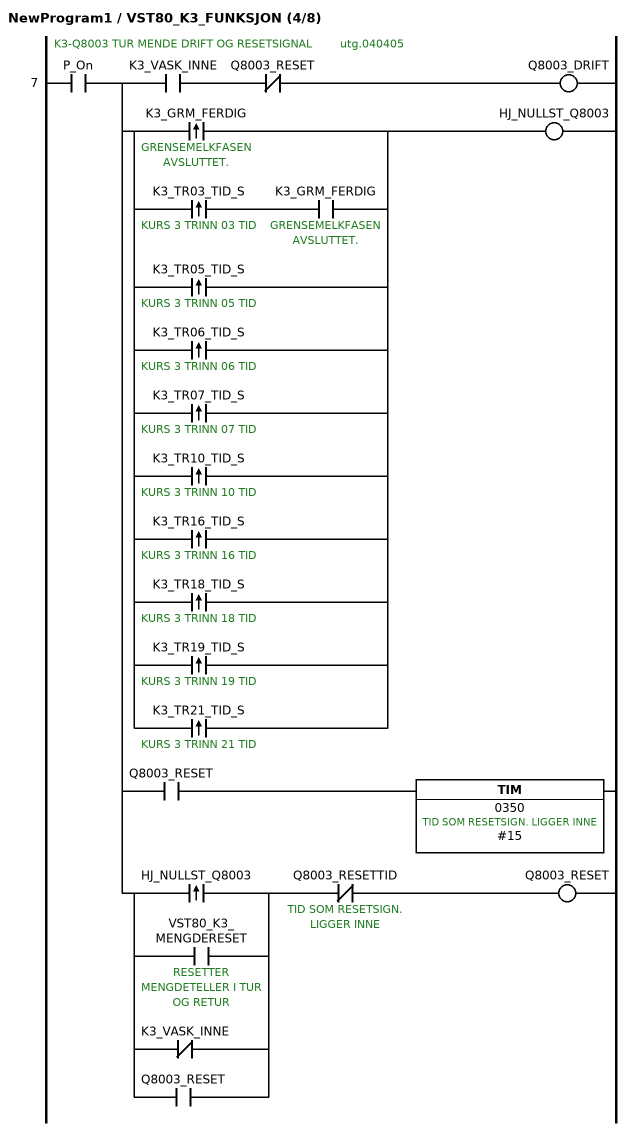
; [picture p360: NewProgram1 / VST80_K3_FUNKSJON, rungs 7-7]
; rung 7: K3-Q8003 TUR MENDE DRIFT OG RESETSIGNAL        utg.040405
LD P_On
OUT TR0
AND K3_VASK_INNE
ANDNOT Q8003_RESET
OUT Q8003_DRIFT
LD TR0
@LD K3_GRM_FERDIG  ; GRENSEMELKFASEN AVSLUTTET.
@LD K3_TR03_TID_S  ; KURS 3 TRINN 03 TID
AND K3_GRM_FERDIG  ; GRENSEMELKFASEN AVSLUTTET.
ORLD
@OR K3_TR05_TID_S  ; KURS 3 TRINN 05 TID
@OR K3_TR06_TID_S  ; KURS 3 TRINN 06 TID
@OR K3_TR07_TID_S  ; KURS 3 TRINN 07 TID
@OR K3_TR10_TID_S  ; KURS 3 TRINN 10 TID
@OR K3_TR16_TID_S  ; KURS 3 TRINN 16 TID
@OR K3_TR18_TID_S  ; KURS 3 TRINN 18 TID
@OR K3_TR19_TID_S  ; KURS 3 TRINN 19 TID
@OR K3_TR21_TID_S  ; KURS 3 TRINN 21 TID
ANDLD
OUT HJ_NULLST_Q8003
LD TR0
AND Q8003_RESET
TIM 0350 #15  ; TID SOM RESETSIGN. LIGGER INNE
LD TR0
@LD HJ_NULLST_Q8003
OR VST80_K3_MENGDERESET  ; RESETTER MENGDETELLER I TUR OG RETUR
ORNOT K3_VASK_INNE
OR Q8003_RESET
ANDLD
ANDNOT Q8003_RESETTID  ; TID SOM RESETSIGN. LIGGER INNE
OUT Q8003_RESET

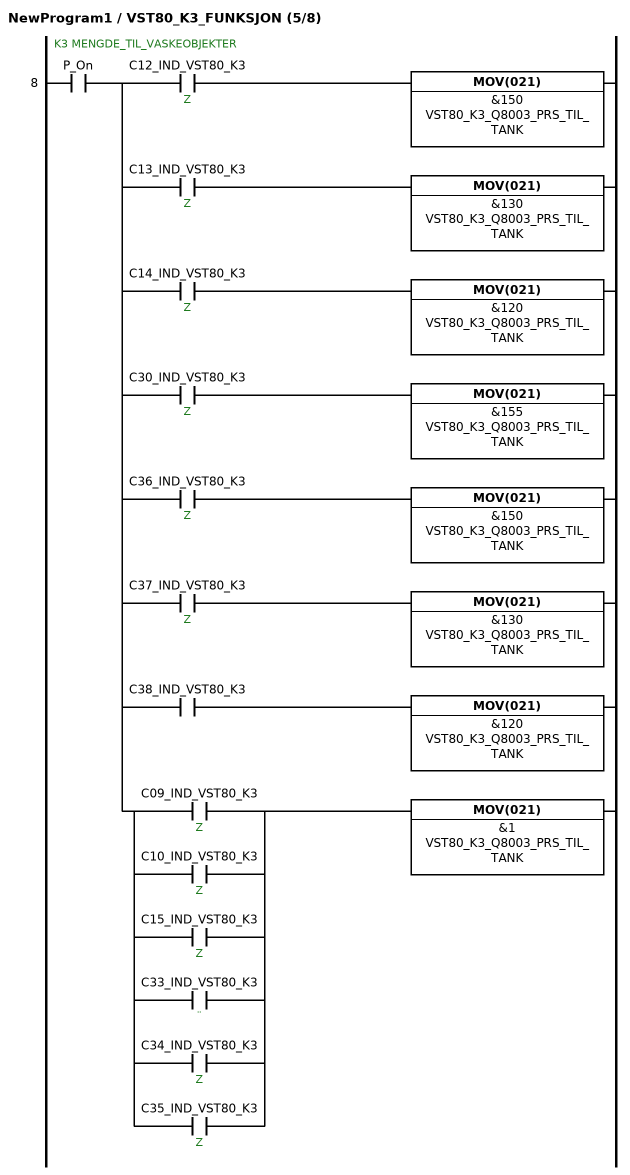
; rung 8: K3 MENGDE_TIL_VASKEOBJEKTER
LD P_On
OUT TR0
AND C12_IND_VST80_K3  ; Z
MOV(021) &150 VST80_K3_Q8003_PRS_TIL_TANK
LD TR0
AND C13_IND_VST80_K3  ; Z
MOV(021) &130 VST80_K3_Q8003_PRS_TIL_TANK
LD TR0
AND C14_IND_VST80_K3  ; Z
MOV(021) &120 VST80_K3_Q8003_PRS_TIL_TANK
LD TR0
AND C30_IND_VST80_K3  ; Z
MOV(021) &155 VST80_K3_Q8003_PRS_TIL_TANK
LD TR0
AND C36_IND_VST80_K3  ; Z
MOV(021) &150 VST80_K3_Q8003_PRS_TIL_TANK
LD TR0
AND C37_IND_VST80_K3  ; Z
MOV(021) &130 VST80_K3_Q8003_PRS_TIL_TANK
LD TR0
AND C38_IND_VST80_K3
MOV(021) &120 VST80_K3_Q8003_PRS_TIL_TANK
LD TR0
LD C09_IND_VST80_K3  ; Z
OR C10_IND_VST80_K3  ; Z
OR C15_IND_VST80_K3  ; Z
OR C33_IND_VST80_K3  ; ¨
OR C34_IND_VST80_K3  ; Z
OR C35_IND_VST80_K3  ; Z
ANDLD
MOV(021) &1 VST80_K3_Q8003_PRS_TIL_TANK

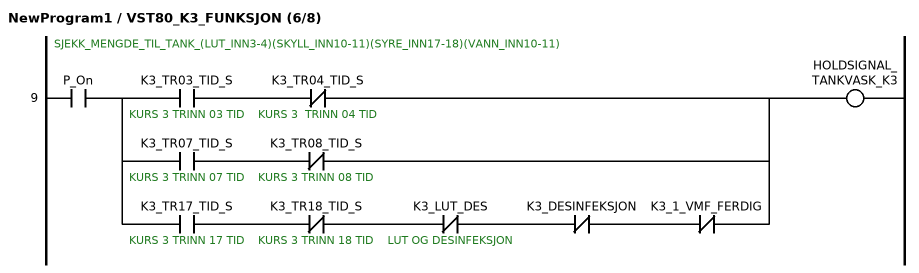
; rung 9: SJEKK_MENGDE_TIL_TANK_(LUT_INN3-4)(SKYLL_INN10-11)(SYRE_INN17-18)(VANN_INN10-11)
LD P_On
LD K3_TR03_TID_S  ; KURS 3 TRINN 03 TID
ANDNOT K3_TR04_TID_S  ; KURS 3  TRINN 04 TID
LD K3_TR07_TID_S  ; KURS 3 TRINN 07 TID
ANDNOT K3_TR08_TID_S  ; KURS 3 TRINN 08 TID
ORLD
LD K3_TR17_TID_S  ; KURS 3 TRINN 17 TID
ANDNOT K3_TR18_TID_S  ; KURS 3 TRINN 18 TID
ANDNOT K3_LUT_DES  ; LUT OG DESINFEKSJON
ANDNOT K3_DESINFEKSJON
ANDNOT K3_1_VMF_FERDIG
ORLD
ANDLD
OUT HOLDSIGNAL_TANKVASK_K3

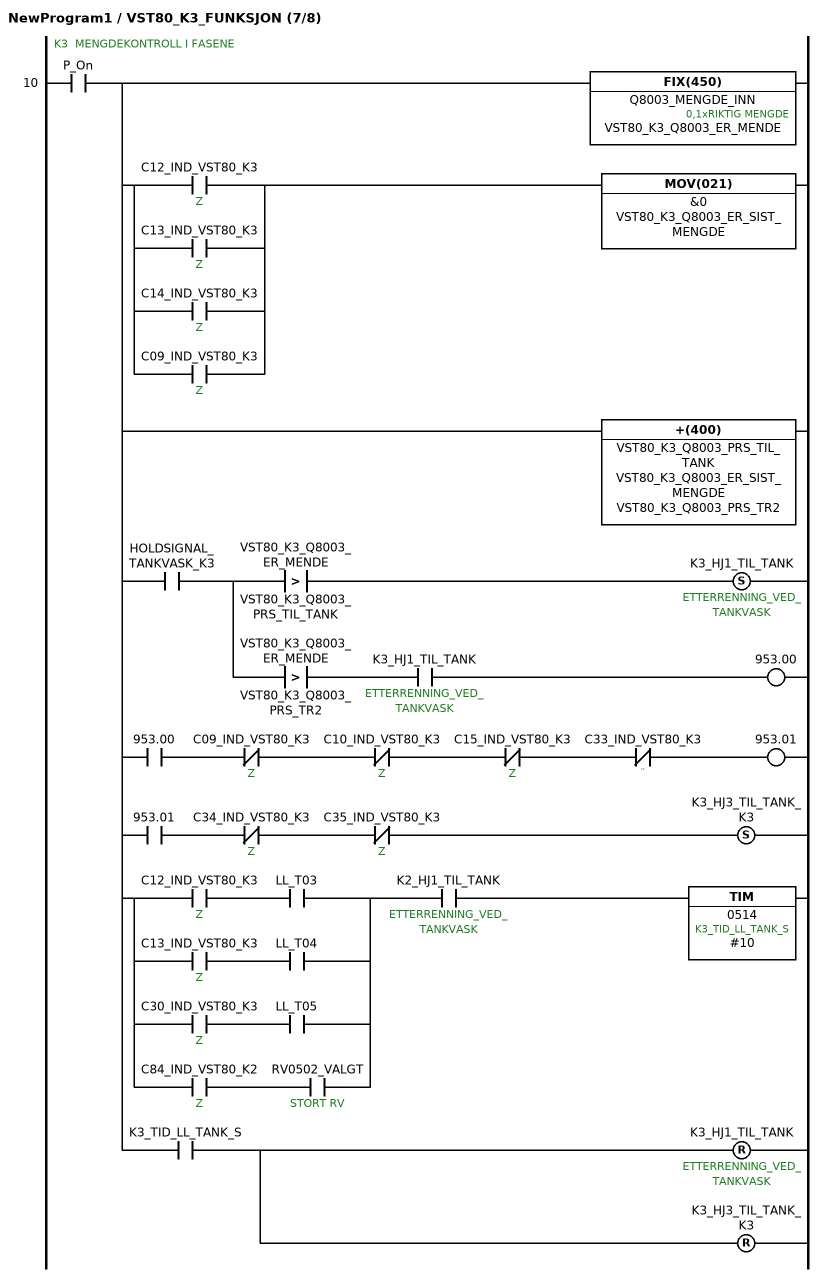
; rung 10: K3  MENGDEKONTROLL I FASENE
LD P_On
OUT TR0
FIX(450) Q8003_MENGDE_INN VST80_K3_Q8003_ER_MENDE  ; 0,1xRIKTIG MENGDE
LD C12_IND_VST80_K3  ; Z
OR C13_IND_VST80_K3  ; Z
OR C14_IND_VST80_K3  ; Z
OR C09_IND_VST80_K3  ; Z
ANDLD
MOV(021) &0 VST80_K3_Q8003_ER_SIST_MENGDE
LD TR0
+(400) VST80_K3_Q8003_PRS_TIL_TANK VST80_K3_Q8003_ER_SIST_MENGDE VST80_K3_Q8003_PRS_TR2
AND HOLDSIGNAL_TANKVASK_K3
OUT TR1
AND>(320) VST80_K3_Q8003_ER_MENDE VST80_K3_Q8003_PRS_TIL_TANK
SET K3_HJ1_TIL_TANK  ; ETTERRENNING_VED_TANKVASK
LD TR1
AND>(320) VST80_K3_Q8003_ER_MENDE VST80_K3_Q8003_PRS_TR2
AND K3_HJ1_TIL_TANK  ; ETTERRENNING_VED_TANKVASK
OUT 953.00
LD TR0
AND 953.00
ANDNOT C09_IND_VST80_K3  ; Z
ANDNOT C10_IND_VST80_K3  ; Z
ANDNOT C15_IND_VST80_K3  ; Z
ANDNOT C33_IND_VST80_K3  ; ¨
OUT 953.01
LD TR0
AND 953.01
ANDNOT C34_IND_VST80_K3  ; Z
ANDNOT C35_IND_VST80_K3  ; Z
SET K3_HJ3_TIL_TANK_K3
LD TR0
LD C12_IND_VST80_K3  ; Z
AND LL_T03
LD C13_IND_VST80_K3  ; Z
AND LL_T04
ORLD
LD C30_IND_VST80_K3  ; Z
AND LL_T05
ORLD
LD C84_IND_VST80_K2  ; Z
AND RV0502_VALGT  ; STORT RV
ORLD
ANDLD
AND K2_HJ1_TIL_TANK  ; ETTERRENNING_VED_TANKVASK
TIM 0514 #10  ; K3_TID_LL_TANK_S
LD TR0
AND K3_TID_LL_TANK_S
RSET K3_HJ1_TIL_TANK  ; ETTERRENNING_VED_TANKVASK
RSET K3_HJ3_TIL_TANK_K3

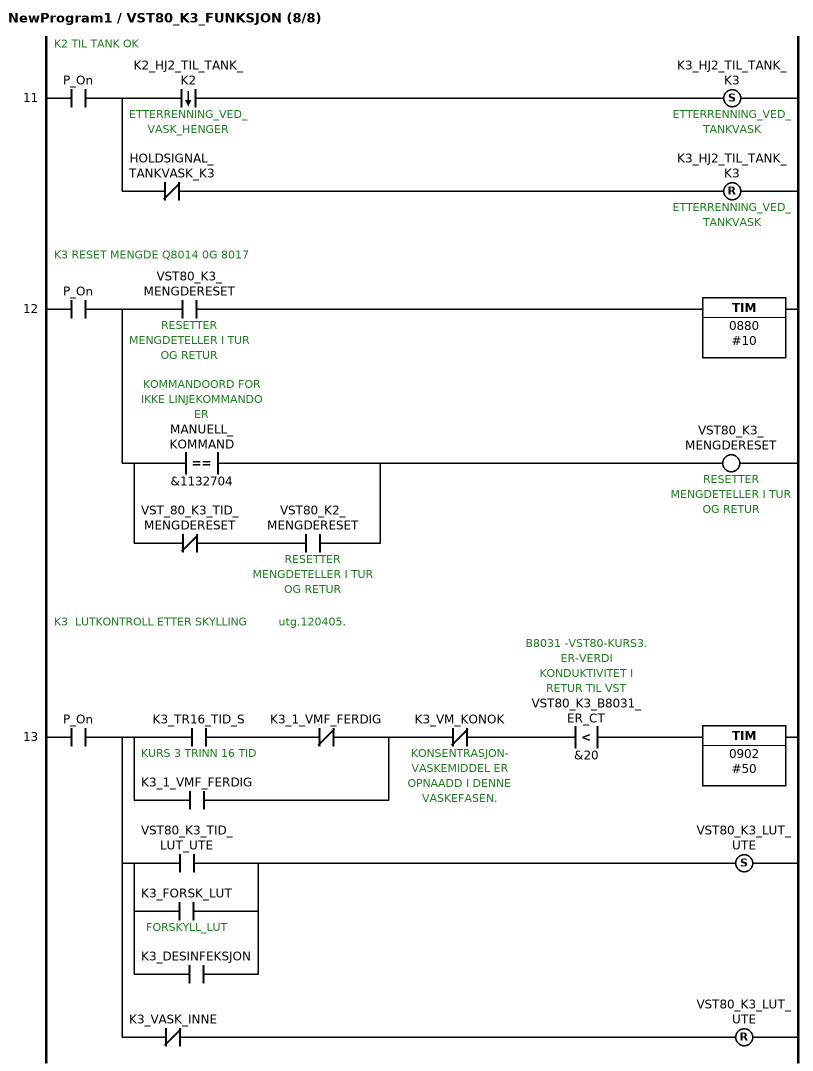
; rung 11: K2 TIL TANK OK
LD P_On
OUT TR0
%AND K2_HJ2_TIL_TANK_K2  ; ETTERRENNING_VED_VASK_HENGER
SET K3_HJ2_TIL_TANK_K3  ; ETTERRENNING_VED_TANKVASK
LD TR0
ANDNOT HOLDSIGNAL_TANKVASK_K3
RSET K3_HJ2_TIL_TANK_K3  ; ETTERRENNING_VED_TANKVASK
; rung 12: K3 RESET MENGDE Q8014 0G 8017
LD P_On
OUT TR0
AND VST80_K3_MENGDERESET  ; RESETTER MENGDETELLER I TUR OG RETUR
TIM 0880 #10
LD TR0
LD=L(301) MANUELL_KOMMAND &1132704  ; KOMMANDOORD FOR IKKE LINJEKOMMANDOER
LDNOT VST_80_K3_TID_MENGDERESET
AND VST80_K2_MENGDERESET  ; RESETTER MENGDETELLER I TUR OG RETUR
ORLD
ANDLD
OUT VST80_K3_MENGDERESET  ; RESETTER MENGDETELLER I TUR OG RETUR
; rung 13: K3  LUTKONTROLL ETTER SKYLLING         utg.120405.
LD P_On
OUT TR0
LD K3_TR16_TID_S  ; KURS 3 TRINN 16 TID
ANDNOT K3_1_VMF_FERDIG
OR K3_1_VMF_FERDIG
ANDLD
ANDNOT K3_VM_KONOK  ; KONSENTRASJON-VASKEMIDDEL ER OPNAADD I DENNE VASKEFASEN.
AND<(310) VST80_K3_B8031_ER_CT &20  ; B8031 -VST80-KURS3. ER-VERDI KONDUKTIVITET I RETUR TIL VST
TIM 0902 #50
LD TR0
LD VST80_K3_TID_LUT_UTE
OR K3_FORSK_LUT  ; FORSKYLL_LUT
OR K3_DESINFEKSJON
ANDLD
SET VST80_K3_LUT_UTE
LD TR0
ANDNOT K3_VASK_INNE
RSET VST80_K3_LUT_UTE
; rung 14: Ingen_kommentar_funnet

### Section VST80_K3_OBJEKTER
; Styring av objektene i kurs K1

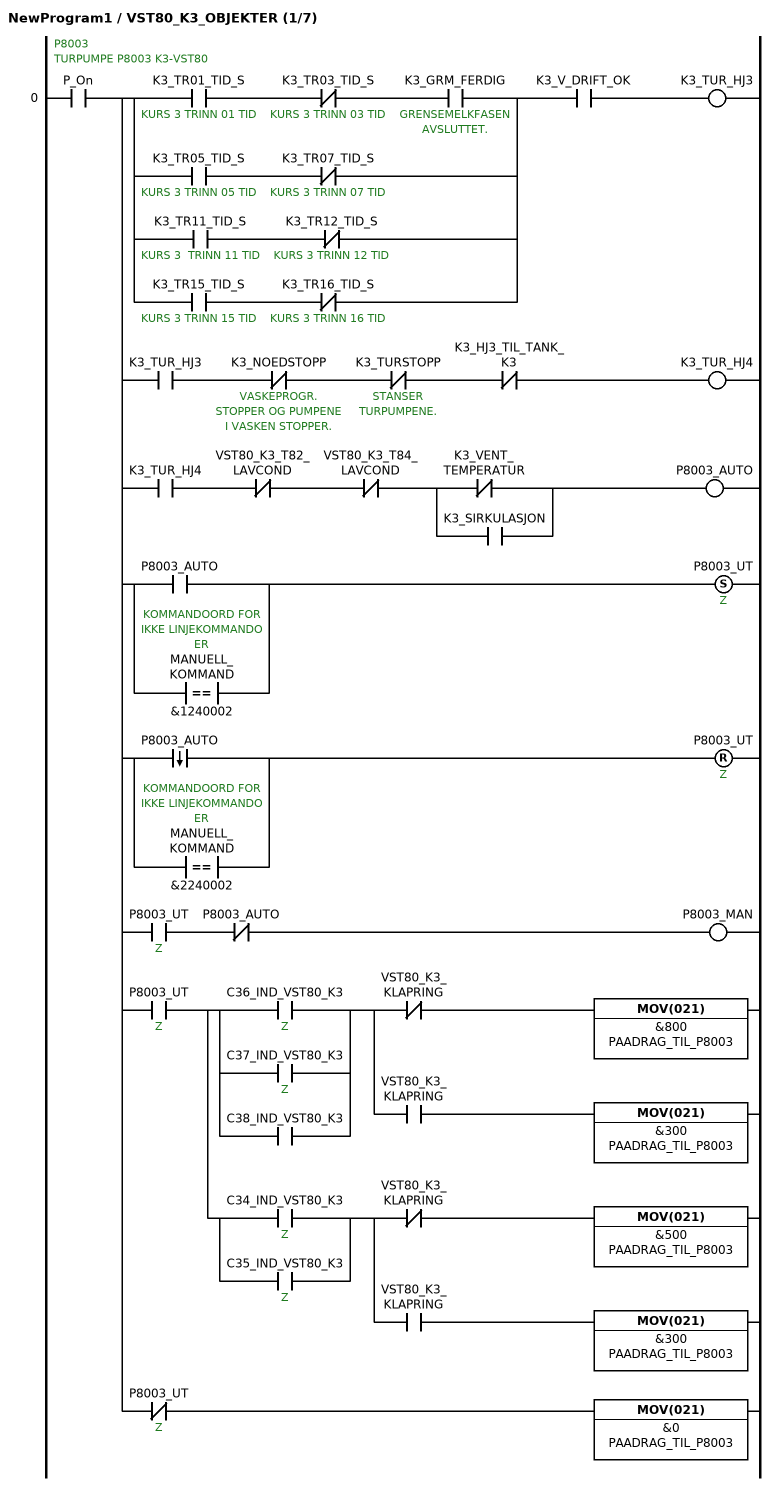
; rung 0: P8003 / TURPUMPE P8003 K3-VST80
LD P_On
OUT TR0
LD K3_TR01_TID_S  ; KURS 3 TRINN 01 TID
ANDNOT K3_TR03_TID_S  ; KURS 3 TRINN 03 TID
AND K3_GRM_FERDIG  ; GRENSEMELKFASEN AVSLUTTET.
LD K3_TR05_TID_S  ; KURS 3 TRINN 05 TID
ANDNOT K3_TR07_TID_S  ; KURS 3 TRINN 07 TID
ORLD
LD K3_TR11_TID_S  ; KURS 3  TRINN 11 TID
ANDNOT K3_TR12_TID_S  ; KURS 3 TRINN 12 TID
ORLD
LD K3_TR15_TID_S  ; KURS 3 TRINN 15 TID
ANDNOT K3_TR16_TID_S  ; KURS 3 TRINN 16 TID
ORLD
ANDLD
AND K3_V_DRIFT_OK
OUT K3_TUR_HJ3
LD TR0
AND K3_TUR_HJ3
ANDNOT K3_NOEDSTOPP  ; VASKEPROGR. STOPPER OG PUMPENE I VASKEN STOPPER.
ANDNOT K3_TURSTOPP  ; STANSER TURPUMPENE.
ANDNOT K3_HJ3_TIL_TANK_K3
OUT K3_TUR_HJ4
LD TR0
AND K3_TUR_HJ4
ANDNOT VST80_K3_T82_LAVCOND
ANDNOT VST80_K3_T84_LAVCOND
LDNOT K3_VENT_TEMPERATUR
OR K3_SIRKULASJON
ANDLD
OUT P8003_AUTO
LD TR0
LD P8003_AUTO
OR=L(301) MANUELL_KOMMAND &1240002  ; KOMMANDOORD FOR IKKE LINJEKOMMANDOER
ANDLD
SET P8003_UT  ; Z
LD TR0
%LD P8003_AUTO
OR=L(301) MANUELL_KOMMAND &2240002  ; KOMMANDOORD FOR IKKE LINJEKOMMANDOER
ANDLD
RSET P8003_UT  ; Z
LD TR0
AND P8003_UT  ; Z
ANDNOT P8003_AUTO
OUT P8003_MAN
LD TR0
AND P8003_UT  ; Z
OUT TR1
LD C36_IND_VST80_K3  ; Z
OR C37_IND_VST80_K3  ; Z
OR C38_IND_VST80_K3
ANDLD
OUT TR2
ANDNOT VST80_K3_KLAPRING
MOV(021) &800 PAADRAG_TIL_P8003
LD TR2
AND VST80_K3_KLAPRING
MOV(021) &300 PAADRAG_TIL_P8003
LD TR1
LD C34_IND_VST80_K3  ; Z
OR C35_IND_VST80_K3  ; Z
ANDLD
OUT TR1
ANDNOT VST80_K3_KLAPRING
MOV(021) &500 PAADRAG_TIL_P8003
LD TR1
AND VST80_K3_KLAPRING
MOV(021) &300 PAADRAG_TIL_P8003
LD TR0
ANDNOT P8003_UT  ; Z
MOV(021) &0 PAADRAG_TIL_P8003

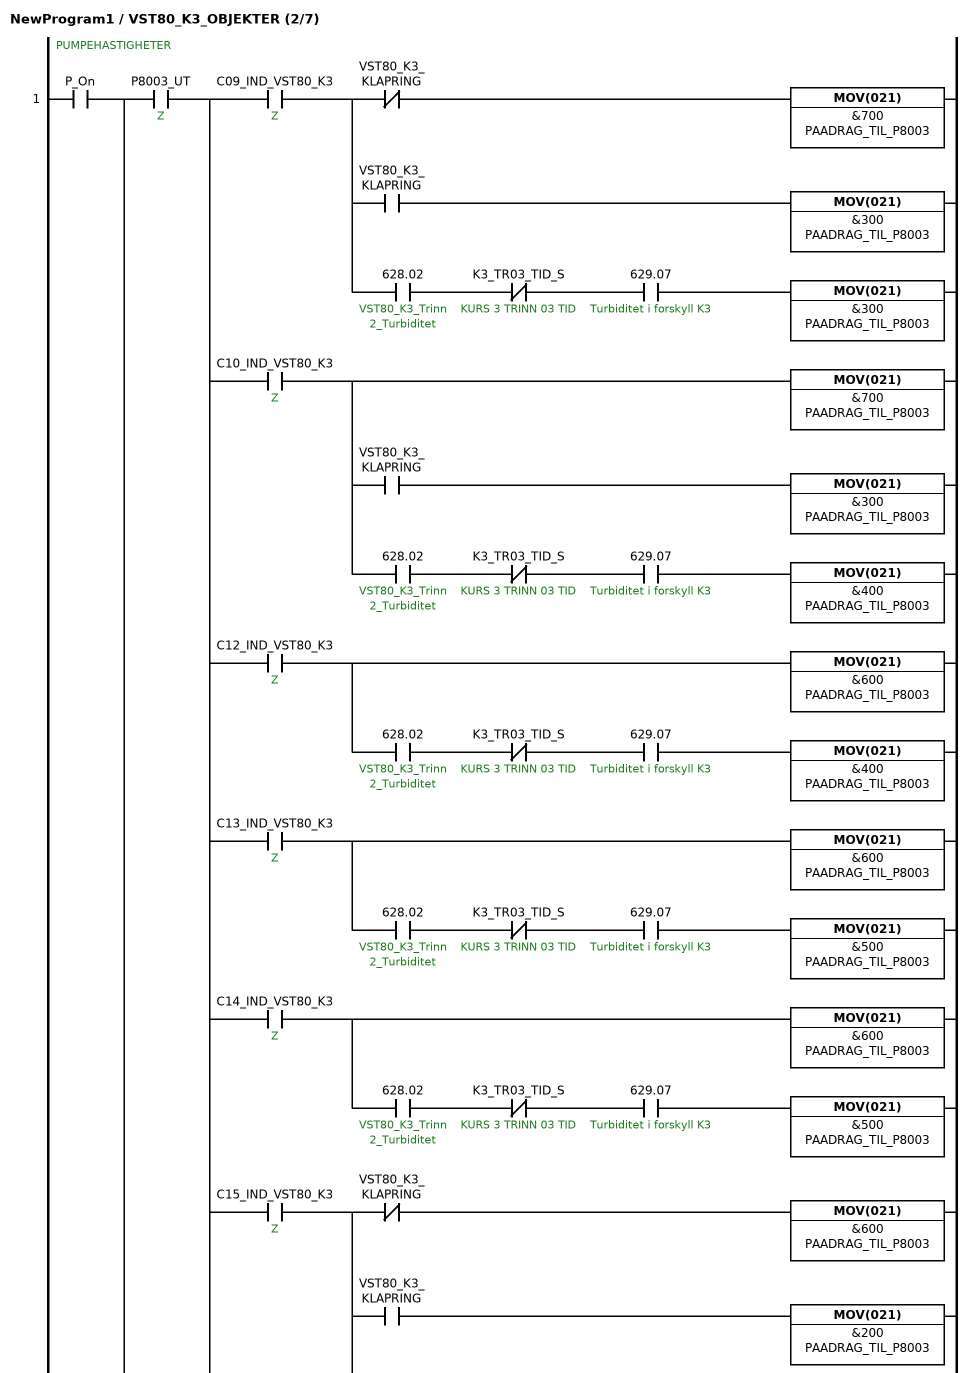

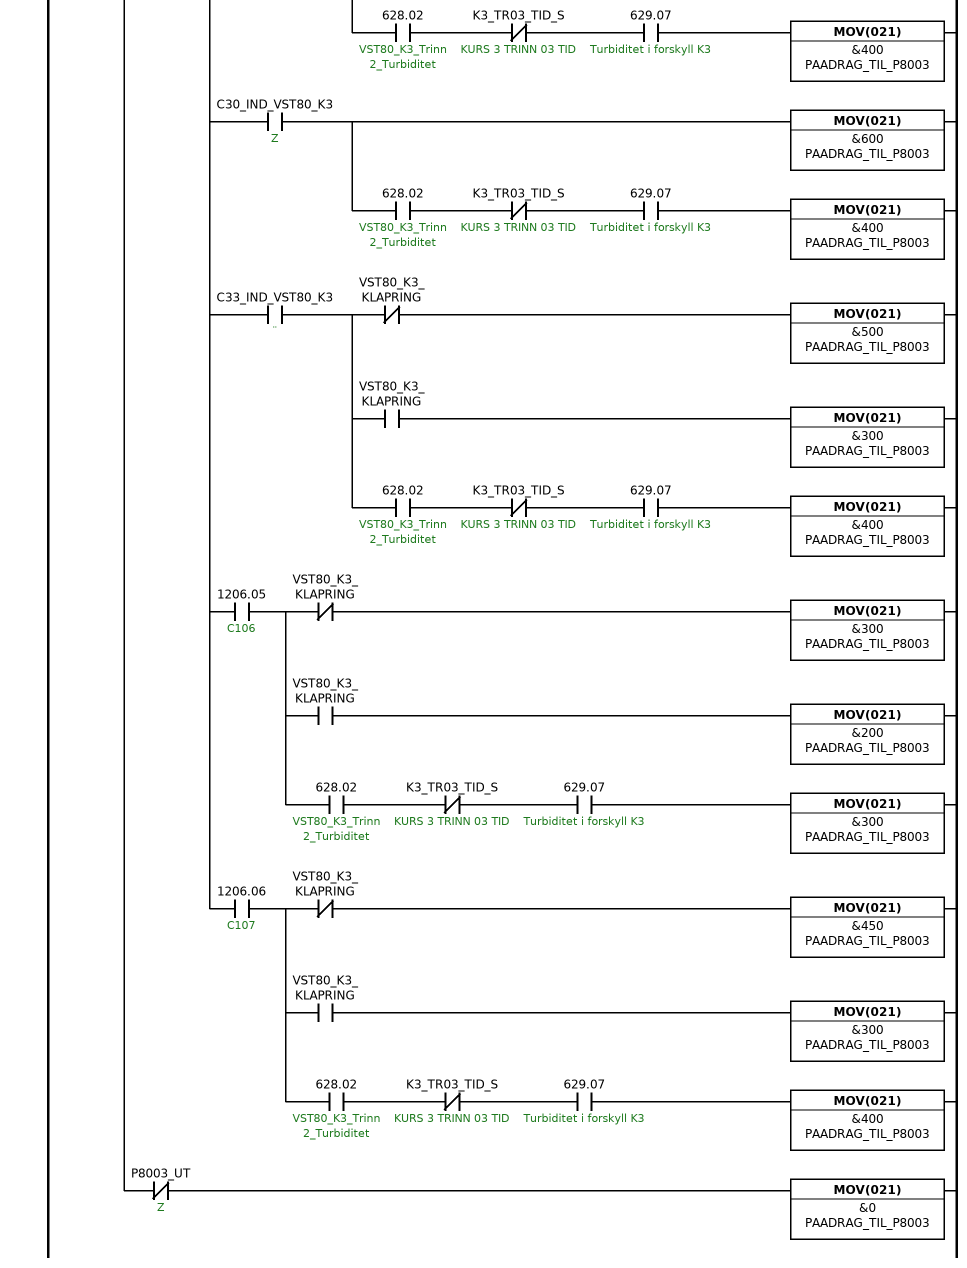
; rung 1: PUMPEHASTIGHETER
LD P_On
OUT TR0
AND P8003_UT  ; Z
OUT TR1
AND C09_IND_VST80_K3  ; Z
OUT TR2
ANDNOT VST80_K3_KLAPRING
MOV(021) &700 PAADRAG_TIL_P8003
LD TR2
AND VST80_K3_KLAPRING
MOV(021) &300 PAADRAG_TIL_P8003
LD TR2
AND 628.02  ; VST80_K3_Trinn 2_Turbiditet
ANDNOT K3_TR03_TID_S  ; KURS 3 TRINN 03 TID
AND 629.07  ; Turbiditet i forskyll K3
MOV(021) &300 PAADRAG_TIL_P8003
LD TR1
AND C10_IND_VST80_K3  ; Z
OUT TR2
MOV(021) &700 PAADRAG_TIL_P8003
AND VST80_K3_KLAPRING
MOV(021) &300 PAADRAG_TIL_P8003
LD TR2
AND 628.02  ; VST80_K3_Trinn 2_Turbiditet
ANDNOT K3_TR03_TID_S  ; KURS 3 TRINN 03 TID
AND 629.07  ; Turbiditet i forskyll K3
MOV(021) &400 PAADRAG_TIL_P8003
LD TR1
AND C12_IND_VST80_K3  ; Z
MOV(021) &600 PAADRAG_TIL_P8003
AND 628.02  ; VST80_K3_Trinn 2_Turbiditet
ANDNOT K3_TR03_TID_S  ; KURS 3 TRINN 03 TID
AND 629.07  ; Turbiditet i forskyll K3
MOV(021) &400 PAADRAG_TIL_P8003
LD TR1
AND C13_IND_VST80_K3  ; Z
MOV(021) &600 PAADRAG_TIL_P8003
AND 628.02  ; VST80_K3_Trinn 2_Turbiditet
ANDNOT K3_TR03_TID_S  ; KURS 3 TRINN 03 TID
AND 629.07  ; Turbiditet i forskyll K3
MOV(021) &500 PAADRAG_TIL_P8003
LD TR1
AND C14_IND_VST80_K3  ; Z
MOV(021) &600 PAADRAG_TIL_P8003
AND 628.02  ; VST80_K3_Trinn 2_Turbiditet
ANDNOT K3_TR03_TID_S  ; KURS 3 TRINN 03 TID
AND 629.07  ; Turbiditet i forskyll K3
MOV(021) &500 PAADRAG_TIL_P8003
LD TR1
AND C15_IND_VST80_K3  ; Z
OUT TR2
ANDNOT VST80_K3_KLAPRING
MOV(021) &600 PAADRAG_TIL_P8003
LD TR2
AND VST80_K3_KLAPRING
MOV(021) &200 PAADRAG_TIL_P8003
LD TR2
AND 628.02  ; VST80_K3_Trinn 2_Turbiditet
ANDNOT K3_TR03_TID_S  ; KURS 3 TRINN 03 TID
AND 629.07  ; Turbiditet i forskyll K3
MOV(021) &400 PAADRAG_TIL_P8003
LD TR1
AND C30_IND_VST80_K3  ; Z
MOV(021) &600 PAADRAG_TIL_P8003
AND 628.02  ; VST80_K3_Trinn 2_Turbiditet
ANDNOT K3_TR03_TID_S  ; KURS 3 TRINN 03 TID
AND 629.07  ; Turbiditet i forskyll K3
MOV(021) &400 PAADRAG_TIL_P8003
LD TR1
AND C33_IND_VST80_K3  ; ¨
OUT TR2
ANDNOT VST80_K3_KLAPRING
MOV(021) &500 PAADRAG_TIL_P8003
LD TR2
AND VST80_K3_KLAPRING
MOV(021) &300 PAADRAG_TIL_P8003
LD TR2
AND 628.02  ; VST80_K3_Trinn 2_Turbiditet
ANDNOT K3_TR03_TID_S  ; KURS 3 TRINN 03 TID
AND 629.07  ; Turbiditet i forskyll K3
MOV(021) &400 PAADRAG_TIL_P8003
LD TR1
AND 1206.05  ; C106
OUT TR2
ANDNOT VST80_K3_KLAPRING
MOV(021) &300 PAADRAG_TIL_P8003
LD TR2
AND VST80_K3_KLAPRING
MOV(021) &200 PAADRAG_TIL_P8003
LD TR2
AND 628.02  ; VST80_K3_Trinn 2_Turbiditet
ANDNOT K3_TR03_TID_S  ; KURS 3 TRINN 03 TID
AND 629.07  ; Turbiditet i forskyll K3
MOV(021) &300 PAADRAG_TIL_P8003
LD TR1
AND 1206.06  ; C107
OUT TR1
ANDNOT VST80_K3_KLAPRING
MOV(021) &450 PAADRAG_TIL_P8003
LD TR1
AND VST80_K3_KLAPRING
MOV(021) &300 PAADRAG_TIL_P8003
LD TR1
AND 628.02  ; VST80_K3_Trinn 2_Turbiditet
ANDNOT K3_TR03_TID_S  ; KURS 3 TRINN 03 TID
AND 629.07  ; Turbiditet i forskyll K3
MOV(021) &400 PAADRAG_TIL_P8003
LD TR0
ANDNOT P8003_UT  ; Z
MOV(021) &0 PAADRAG_TIL_P8003

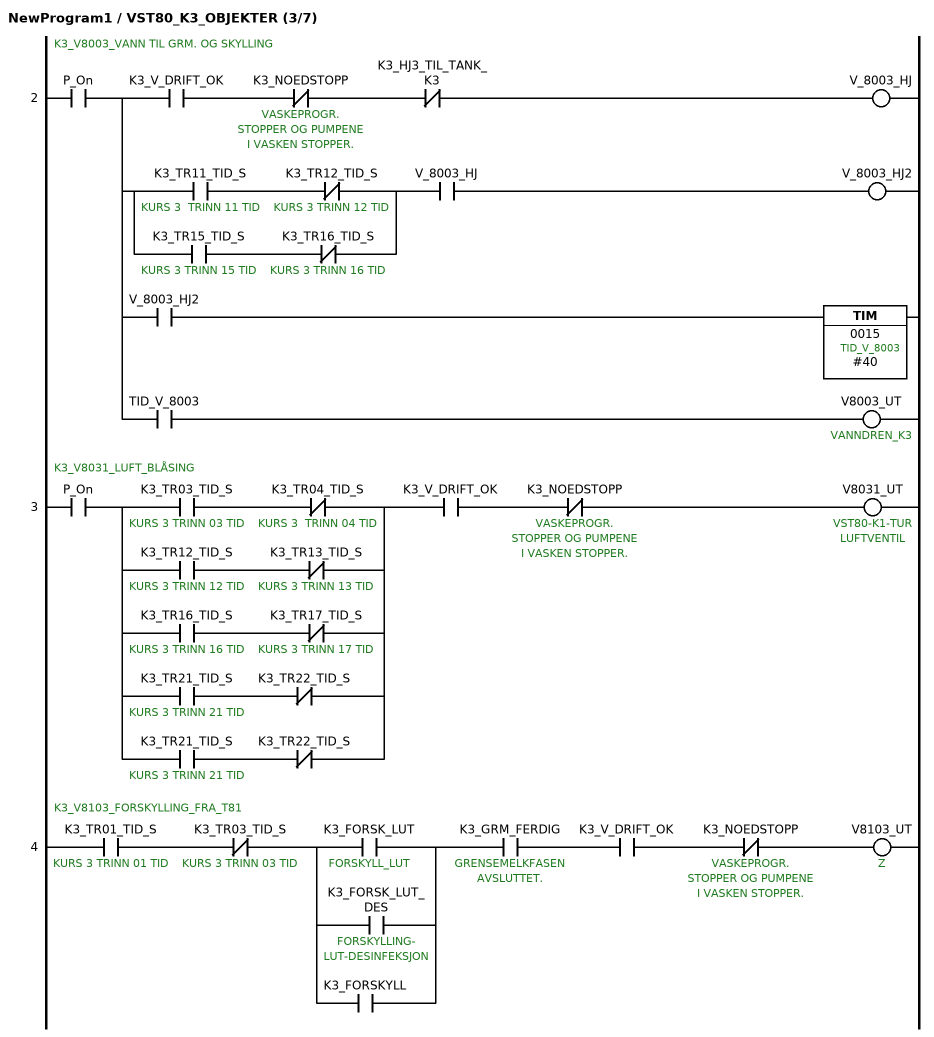
; rung 2: K3_V8003_VANN TIL GRM. OG SKYLLING
LD P_On
OUT TR0
AND K3_V_DRIFT_OK
ANDNOT K3_NOEDSTOPP  ; VASKEPROGR. STOPPER OG PUMPENE I VASKEN STOPPER.
ANDNOT K3_HJ3_TIL_TANK_K3
OUT V_8003_HJ
LD TR0
LD K3_TR11_TID_S  ; KURS 3  TRINN 11 TID
ANDNOT K3_TR12_TID_S  ; KURS 3 TRINN 12 TID
LD K3_TR15_TID_S  ; KURS 3 TRINN 15 TID
ANDNOT K3_TR16_TID_S  ; KURS 3 TRINN 16 TID
ORLD
ANDLD
AND V_8003_HJ
OUT V_8003_HJ2
LD TR0
AND V_8003_HJ2
TIM 0015 #40  ; TID_V_8003
LD TR0
AND TID_V_8003
OUT V8003_UT  ; VANNDREN_K3
; rung 3: K3_V8031_LUFT_BLÅSING
LD P_On
LD K3_TR03_TID_S  ; KURS 3 TRINN 03 TID
ANDNOT K3_TR04_TID_S  ; KURS 3  TRINN 04 TID
LD K3_TR12_TID_S  ; KURS 3 TRINN 12 TID
ANDNOT K3_TR13_TID_S  ; KURS 3 TRINN 13 TID
ORLD
LD K3_TR16_TID_S  ; KURS 3 TRINN 16 TID
ANDNOT K3_TR17_TID_S  ; KURS 3 TRINN 17 TID
ORLD
LD K3_TR21_TID_S  ; KURS 3 TRINN 21 TID
ANDNOT K3_TR22_TID_S
ORLD
LD K3_TR21_TID_S  ; KURS 3 TRINN 21 TID
ANDNOT K3_TR22_TID_S
ORLD
ANDLD
AND K3_V_DRIFT_OK
ANDNOT K3_NOEDSTOPP  ; VASKEPROGR. STOPPER OG PUMPENE I VASKEN STOPPER.
OUT V8031_UT  ; VST80-K1-TUR LUFTVENTIL
; rung 4: K3_V8103_FORSKYLLING_FRA_T81
LD K3_TR01_TID_S  ; KURS 3 TRINN 01 TID
ANDNOT K3_TR03_TID_S  ; KURS 3 TRINN 03 TID
LD K3_FORSK_LUT  ; FORSKYLL_LUT
OR K3_FORSK_LUT_DES  ; FORSKYLLING- LUT-DESINFEKSJON
OR K3_FORSKYLL
ANDLD
AND K3_GRM_FERDIG  ; GRENSEMELKFASEN AVSLUTTET.
AND K3_V_DRIFT_OK
ANDNOT K3_NOEDSTOPP  ; VASKEPROGR. STOPPER OG PUMPENE I VASKEN STOPPER.
OUT V8103_UT  ; Z

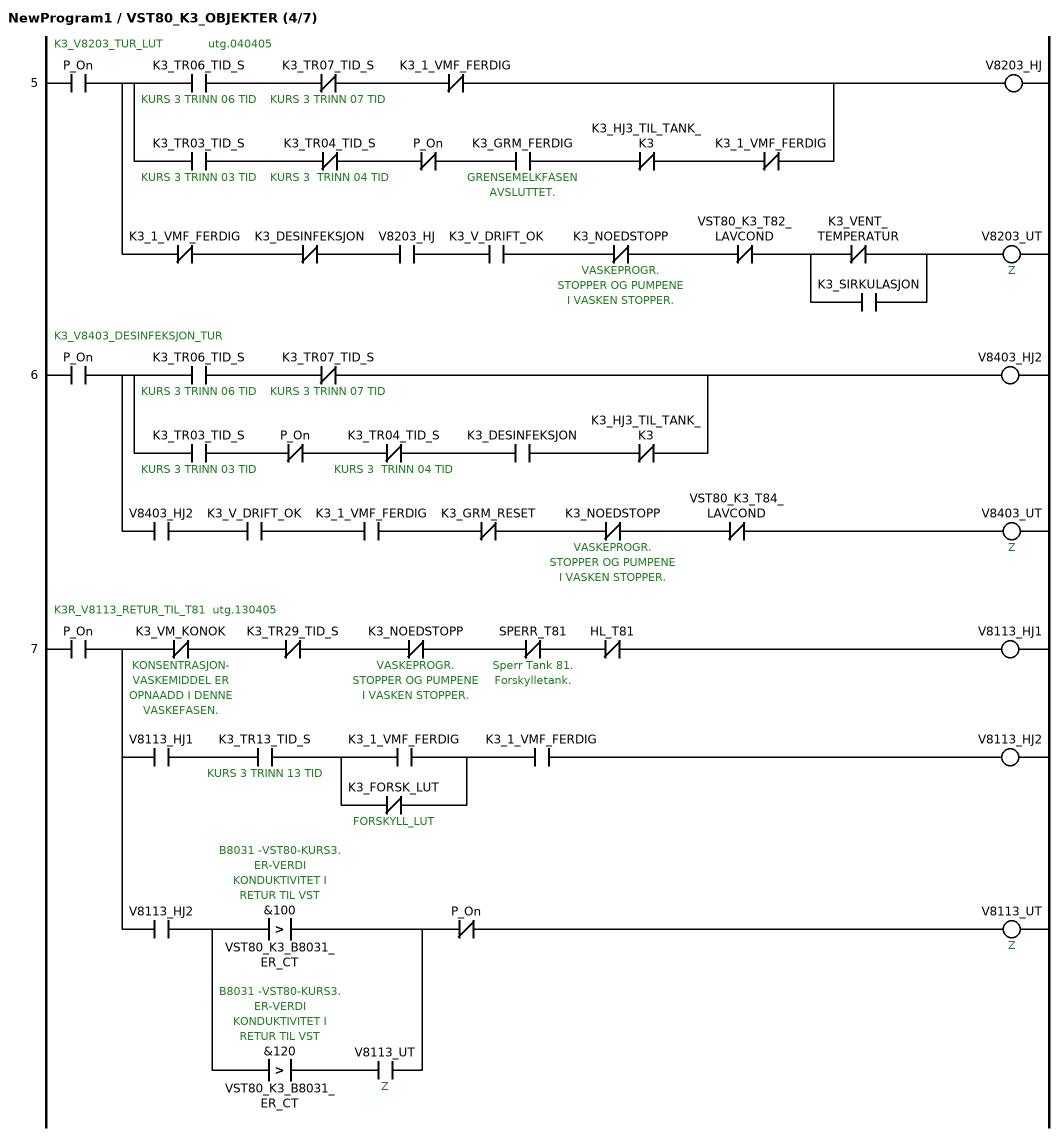
; rung 5: K3_V8203_TUR_LUT             utg.040405
LD P_On
OUT TR0
LD K3_TR06_TID_S  ; KURS 3 TRINN 06 TID
ANDNOT K3_TR07_TID_S  ; KURS 3 TRINN 07 TID
ANDNOT K3_1_VMF_FERDIG
LD K3_TR03_TID_S  ; KURS 3 TRINN 03 TID
ANDNOT K3_TR04_TID_S  ; KURS 3  TRINN 04 TID
ANDNOT P_On
AND K3_GRM_FERDIG  ; GRENSEMELKFASEN AVSLUTTET.
ANDNOT K3_HJ3_TIL_TANK_K3
ANDNOT K3_1_VMF_FERDIG
ORLD
ANDLD
OUT V8203_HJ
LD TR0
ANDNOT K3_1_VMF_FERDIG
ANDNOT K3_DESINFEKSJON
AND V8203_HJ
AND K3_V_DRIFT_OK
ANDNOT K3_NOEDSTOPP  ; VASKEPROGR. STOPPER OG PUMPENE I VASKEN STOPPER.
ANDNOT VST80_K3_T82_LAVCOND
LDNOT K3_VENT_TEMPERATUR
OR K3_SIRKULASJON
ANDLD
OUT V8203_UT  ; Z
; rung 6: K3_V8403_DESINFEKSJON_TUR
LD P_On
OUT TR0
LD K3_TR06_TID_S  ; KURS 3 TRINN 06 TID
ANDNOT K3_TR07_TID_S  ; KURS 3 TRINN 07 TID
LD K3_TR03_TID_S  ; KURS 3 TRINN 03 TID
ANDNOT P_On
ANDNOT K3_TR04_TID_S  ; KURS 3  TRINN 04 TID
AND K3_DESINFEKSJON
ANDNOT K3_HJ3_TIL_TANK_K3
ORLD
ANDLD
OUT V8403_HJ2
LD TR0
AND V8403_HJ2
AND K3_V_DRIFT_OK
AND K3_1_VMF_FERDIG
ANDNOT K3_GRM_RESET
ANDNOT K3_NOEDSTOPP  ; VASKEPROGR. STOPPER OG PUMPENE I VASKEN STOPPER.
ANDNOT VST80_K3_T84_LAVCOND
OUT V8403_UT  ; Z
; rung 7: K3R_V8113_RETUR_TIL_T81  utg.130405
LD P_On
OUT TR0
ANDNOT K3_VM_KONOK  ; KONSENTRASJON-VASKEMIDDEL ER OPNAADD I DENNE VASKEFASEN.
ANDNOT K3_TR29_TID_S
ANDNOT K3_NOEDSTOPP  ; VASKEPROGR. STOPPER OG PUMPENE I VASKEN STOPPER.
ANDNOT SPERR_T81  ; Sperr Tank 81. Forskylletank.
ANDNOT HL_T81
OUT V8113_HJ1
LD TR0
AND V8113_HJ1
AND K3_TR13_TID_S  ; KURS 3 TRINN 13 TID
LD K3_1_VMF_FERDIG
ORNOT K3_FORSK_LUT  ; FORSKYLL_LUT
ANDLD
AND K3_1_VMF_FERDIG
OUT V8113_HJ2
LD TR0
AND V8113_HJ2
LD>(320) &100 VST80_K3_B8031_ER_CT  ; B8031 -VST80-KURS3. ER-VERDI KONDUKTIVITET I RETUR TIL VST
LD>(320) &120 VST80_K3_B8031_ER_CT  ; B8031 -VST80-KURS3. ER-VERDI KONDUKTIVITET I RETUR TIL VST
AND V8113_UT  ; Z
ORLD
ANDLD
ANDNOT P_On
OUT V8113_UT  ; Z

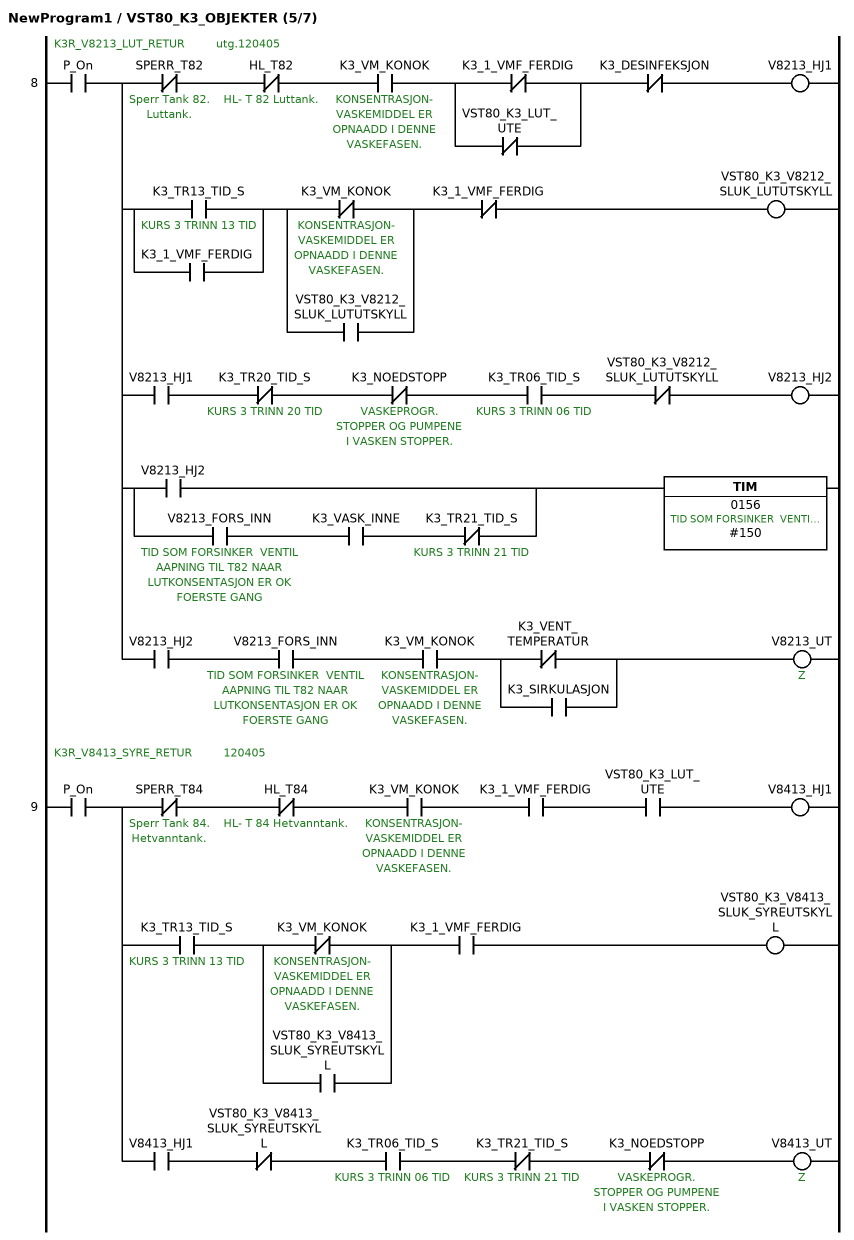
; rung 8: K3R_V8213_LUT_RETUR         utg.120405
LD P_On
OUT TR0
ANDNOT SPERR_T82  ; Sperr Tank 82. Luttank.
ANDNOT HL_T82  ; HL- T 82 Luttank.
AND K3_VM_KONOK  ; KONSENTRASJON-VASKEMIDDEL ER OPNAADD I DENNE VASKEFASEN.
LDNOT K3_1_VMF_FERDIG
ORNOT VST80_K3_LUT_UTE
ANDLD
ANDNOT K3_DESINFEKSJON
OUT V8213_HJ1
LD TR0
LD K3_TR13_TID_S  ; KURS 3 TRINN 13 TID
OR K3_1_VMF_FERDIG
ANDLD
LDNOT K3_VM_KONOK  ; KONSENTRASJON-VASKEMIDDEL ER OPNAADD I DENNE VASKEFASEN.
OR VST80_K3_V8212_SLUK_LUTUTSKYLL
ANDLD
ANDNOT K3_1_VMF_FERDIG
OUT VST80_K3_V8212_SLUK_LUTUTSKYLL
LD TR0
AND V8213_HJ1
ANDNOT K3_TR20_TID_S  ; KURS 3 TRINN 20 TID
ANDNOT K3_NOEDSTOPP  ; VASKEPROGR. STOPPER OG PUMPENE I VASKEN STOPPER.
AND K3_TR06_TID_S  ; KURS 3 TRINN 06 TID
ANDNOT VST80_K3_V8212_SLUK_LUTUTSKYLL
OUT V8213_HJ2
LD TR0
LD V8213_HJ2
LD V8213_FORS_INN  ; TID SOM FORSINKER  VENTIL AAPNING TIL T82 NAAR LUTKONSENTASJON ER OK FOERSTE GANG
AND K3_VASK_INNE
ANDNOT K3_TR21_TID_S  ; KURS 3 TRINN 21 TID
ORLD
ANDLD
TIM 0156 #150  ; TID SOM FORSINKER  VENTIL AAPNING TIL T82 NAAR LUTKONSENTASJON ER OK FOERSTE GANG
LD TR0
AND V8213_HJ2
AND V8213_FORS_INN  ; TID SOM FORSINKER  VENTIL AAPNING TIL T82 NAAR LUTKONSENTASJON ER OK FOERSTE GANG
AND K3_VM_KONOK  ; KONSENTRASJON-VASKEMIDDEL ER OPNAADD I DENNE VASKEFASEN.
LDNOT K3_VENT_TEMPERATUR
OR K3_SIRKULASJON
ANDLD
OUT V8213_UT  ; Z
; rung 9: K3R_V8413_SYRE_RETUR         120405
LD P_On
OUT TR0
ANDNOT SPERR_T84  ; Sperr Tank 84. Hetvanntank.
ANDNOT HL_T84  ; HL- T 84 Hetvanntank.
AND K3_VM_KONOK  ; KONSENTRASJON-VASKEMIDDEL ER OPNAADD I DENNE VASKEFASEN.
AND K3_1_VMF_FERDIG
AND VST80_K3_LUT_UTE
OUT V8413_HJ1
LD TR0
AND K3_TR13_TID_S  ; KURS 3 TRINN 13 TID
LDNOT K3_VM_KONOK  ; KONSENTRASJON-VASKEMIDDEL ER OPNAADD I DENNE VASKEFASEN.
OR VST80_K3_V8413_SLUK_SYREUTSKYLL
ANDLD
AND K3_1_VMF_FERDIG
OUT VST80_K3_V8413_SLUK_SYREUTSKYLL
LD TR0
AND V8413_HJ1
ANDNOT VST80_K3_V8413_SLUK_SYREUTSKYLL
AND K3_TR06_TID_S  ; KURS 3 TRINN 06 TID
ANDNOT K3_TR21_TID_S  ; KURS 3 TRINN 21 TID
ANDNOT K3_NOEDSTOPP  ; VASKEPROGR. STOPPER OG PUMPENE I VASKEN STOPPER.
OUT V8413_UT  ; Z

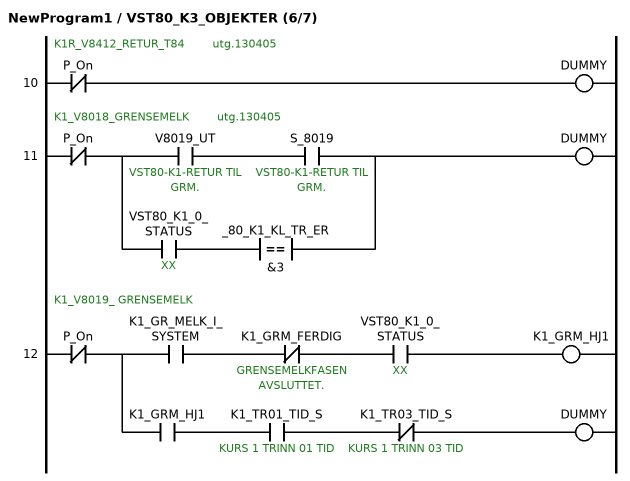
; rung 10: K1R_V8412_RETUR_T84        utg.130405
LDNOT P_On
OUT DUMMY
; rung 11: K1_V8018_GRENSEMELK        utg.130405
LDNOT P_On
LD V8019_UT  ; VST80-K1-RETUR TIL GRM.
AND S_8019  ; VST80-K1-RETUR TIL GRM.
LD VST80_K1_0_STATUS  ; XX
AND=(300) _80_K1_KL_TR_ER &3
ORLD
ANDLD
OUT DUMMY
; rung 12: K1_V8019_GRENSEMELK
LDNOT P_On
OUT TR0
AND K1_GR_MELK_I_SYSTEM
ANDNOT K1_GRM_FERDIG  ; GRENSEMELKFASEN AVSLUTTET.
AND VST80_K1_0_STATUS  ; XX
OUT K1_GRM_HJ1
LD TR0
AND K1_GRM_HJ1
AND K1_TR01_TID_S  ; KURS 1 TRINN 01 TID
ANDNOT K1_TR03_TID_S  ; KURS 1 TRINN 03 TID
OUT DUMMY

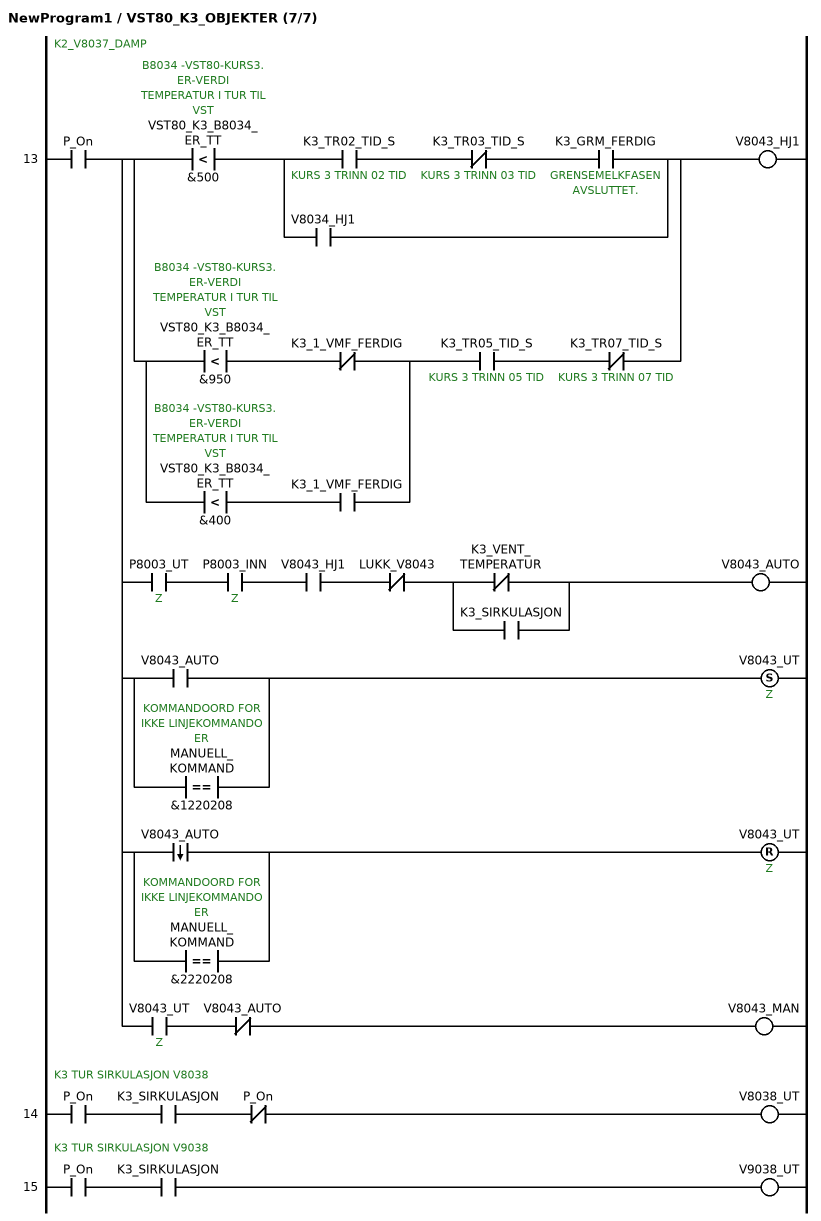
; rung 13: K2_V8037_DAMP
LD P_On
OUT TR0
LD<(310) VST80_K3_B8034_ER_TT &500  ; B8034 -VST80-KURS3. ER-VERDI TEMPERATUR I TUR TIL VST
LD K3_TR02_TID_S  ; KURS 3 TRINN 02 TID
ANDNOT K3_TR03_TID_S  ; KURS 3 TRINN 03 TID
AND K3_GRM_FERDIG  ; GRENSEMELKFASEN AVSLUTTET.
OR V8034_HJ1
ANDLD
LD<(310) VST80_K3_B8034_ER_TT &950  ; B8034 -VST80-KURS3. ER-VERDI TEMPERATUR I TUR TIL VST
ANDNOT K3_1_VMF_FERDIG
LD<(310) VST80_K3_B8034_ER_TT &400  ; B8034 -VST80-KURS3. ER-VERDI TEMPERATUR I TUR TIL VST
AND K3_1_VMF_FERDIG
ORLD
AND K3_TR05_TID_S  ; KURS 3 TRINN 05 TID
ANDNOT K3_TR07_TID_S  ; KURS 3 TRINN 07 TID
ORLD
ANDLD
OUT V8043_HJ1
LD TR0
AND P8003_UT  ; Z
AND P8003_INN  ; Z
AND V8043_HJ1
ANDNOT LUKK_V8043
LDNOT K3_VENT_TEMPERATUR
OR K3_SIRKULASJON
ANDLD
OUT V8043_AUTO
LD TR0
LD V8043_AUTO
OR=L(301) MANUELL_KOMMAND &1220208  ; KOMMANDOORD FOR IKKE LINJEKOMMANDOER
ANDLD
SET V8043_UT  ; Z
LD TR0
%LD V8043_AUTO
OR=L(301) MANUELL_KOMMAND &2220208  ; KOMMANDOORD FOR IKKE LINJEKOMMANDOER
ANDLD
RSET V8043_UT  ; Z
LD TR0
AND V8043_UT  ; Z
ANDNOT V8043_AUTO
OUT V8043_MAN
; rung 14: K3 TUR SIRKULASJON V8038
LD P_On
AND K3_SIRKULASJON
ANDNOT P_On
OUT V8038_UT
; rung 15: K3 TUR SIRKULASJON V9038
LD P_On
AND K3_SIRKULASJON
OUT V9038_UT
; rung 16: Ingen_kommentar_funnet

### Section VST80_K3_KLAPRING
; VST80-KURS1 KLAPREPROGRAM

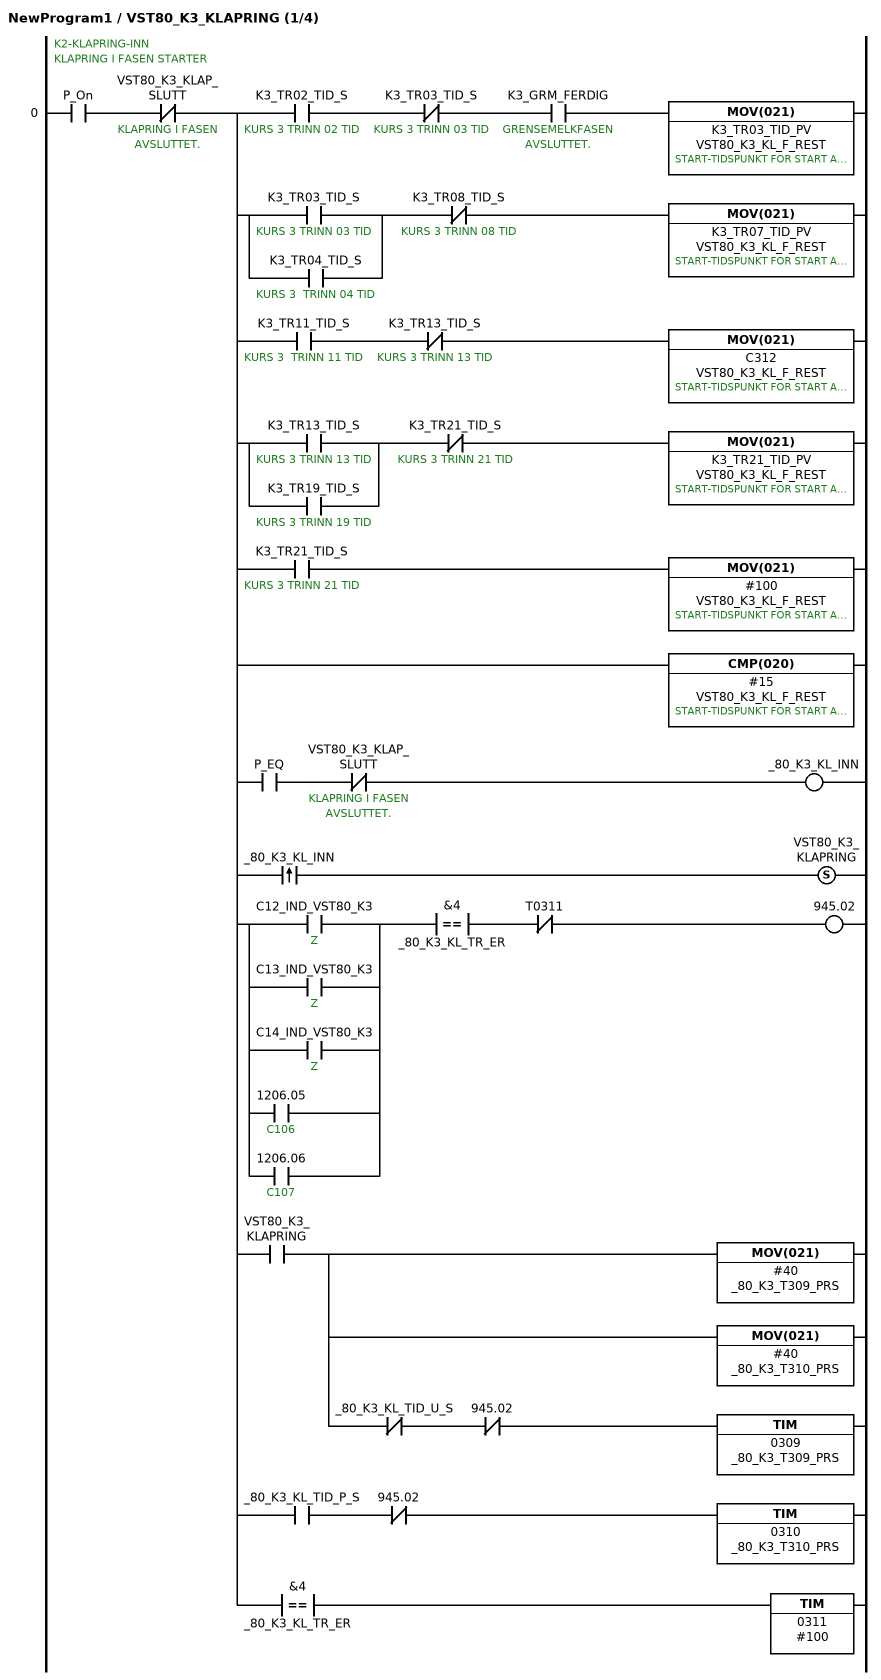
; rung 0: K2-KLAPRING-INN / KLAPRING I FASEN STARTER
LD P_On
ANDNOT VST80_K3_KLAP_SLUTT  ; KLAPRING I FASEN AVSLUTTET.
OUT TR0
AND K3_TR02_TID_S  ; KURS 3 TRINN 02 TID
ANDNOT K3_TR03_TID_S  ; KURS 3 TRINN 03 TID
AND K3_GRM_FERDIG  ; GRENSEMELKFASEN AVSLUTTET.
MOV(021) K3_TR03_TID_PV VST80_K3_KL_F_REST  ; START-TIDSPUNKT FOR START AV KLAPRING
LD TR0
LD K3_TR03_TID_S  ; KURS 3 TRINN 03 TID
OR K3_TR04_TID_S  ; KURS 3  TRINN 04 TID
ANDLD
ANDNOT K3_TR08_TID_S  ; KURS 3 TRINN 08 TID
MOV(021) K3_TR07_TID_PV VST80_K3_KL_F_REST  ; START-TIDSPUNKT FOR START AV KLAPRING
LD TR0
AND K3_TR11_TID_S  ; KURS 3  TRINN 11 TID
ANDNOT K3_TR13_TID_S  ; KURS 3 TRINN 13 TID
MOV(021) C312 VST80_K3_KL_F_REST  ; START-TIDSPUNKT FOR START AV KLAPRING
LD TR0
LD K3_TR13_TID_S  ; KURS 3 TRINN 13 TID
OR K3_TR19_TID_S  ; KURS 3 TRINN 19 TID
ANDLD
ANDNOT K3_TR21_TID_S  ; KURS 3 TRINN 21 TID
MOV(021) K3_TR21_TID_PV VST80_K3_KL_F_REST  ; START-TIDSPUNKT FOR START AV KLAPRING
LD TR0
AND K3_TR21_TID_S  ; KURS 3 TRINN 21 TID
MOV(021) #100 VST80_K3_KL_F_REST  ; START-TIDSPUNKT FOR START AV KLAPRING
LD TR0
CMP(020) #15 VST80_K3_KL_F_REST  ; START-TIDSPUNKT FOR START AV KLAPRING
AND P_EQ
ANDNOT VST80_K3_KLAP_SLUTT  ; KLAPRING I FASEN AVSLUTTET.
OUT _80_K3_KL_INN
LD TR0
@AND _80_K3_KL_INN
SET VST80_K3_KLAPRING
LD TR0
LD C12_IND_VST80_K3  ; Z
OR C13_IND_VST80_K3  ; Z
OR C14_IND_VST80_K3  ; Z
OR 1206.05  ; C106
OR 1206.06  ; C107
ANDLD
AND=(300) &4 _80_K3_KL_TR_ER
ANDNOT T0311
OUT 945.02
LD TR0
AND VST80_K3_KLAPRING
MOV(021) #40 _80_K3_T309_PRS
MOV(021) #40 _80_K3_T310_PRS
ANDNOT _80_K3_KL_TID_U_S
ANDNOT 945.02
TIM 0309 _80_K3_T309_PRS
LD TR0
AND _80_K3_KL_TID_P_S
ANDNOT 945.02
TIM 0310 _80_K3_T310_PRS
LD TR0
AND=(300) &4 _80_K3_KL_TR_ER
TIM 0311 #100

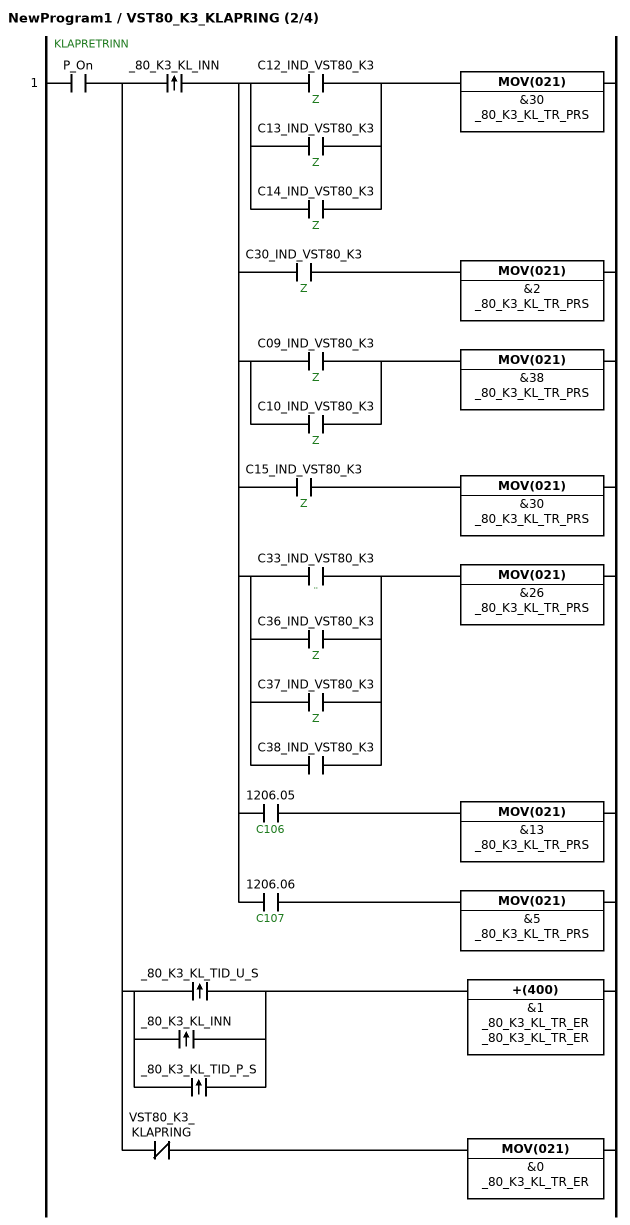
; rung 1: KLAPRETRINN
LD P_On
OUT TR0
@AND _80_K3_KL_INN
OUT TR1
LD C12_IND_VST80_K3  ; Z
OR C13_IND_VST80_K3  ; Z
OR C14_IND_VST80_K3  ; Z
ANDLD
MOV(021) &30 _80_K3_KL_TR_PRS
LD TR1
AND C30_IND_VST80_K3  ; Z
MOV(021) &2 _80_K3_KL_TR_PRS
LD TR1
LD C09_IND_VST80_K3  ; Z
OR C10_IND_VST80_K3  ; Z
ANDLD
MOV(021) &38 _80_K3_KL_TR_PRS
LD TR1
AND C15_IND_VST80_K3  ; Z
MOV(021) &30 _80_K3_KL_TR_PRS
LD TR1
LD C33_IND_VST80_K3  ; ¨
OR C36_IND_VST80_K3  ; Z
OR C37_IND_VST80_K3  ; Z
OR C38_IND_VST80_K3
ANDLD
MOV(021) &26 _80_K3_KL_TR_PRS
LD TR1
AND 1206.05  ; C106
MOV(021) &13 _80_K3_KL_TR_PRS
LD TR1
AND 1206.06  ; C107
MOV(021) &5 _80_K3_KL_TR_PRS
LD TR0
@LD _80_K3_KL_TID_U_S
@OR _80_K3_KL_INN
@OR _80_K3_KL_TID_P_S
ANDLD
+(400) &1 _80_K3_KL_TR_ER _80_K3_KL_TR_ER
LD TR0
ANDNOT VST80_K3_KLAPRING
MOV(021) &0 _80_K3_KL_TR_ER

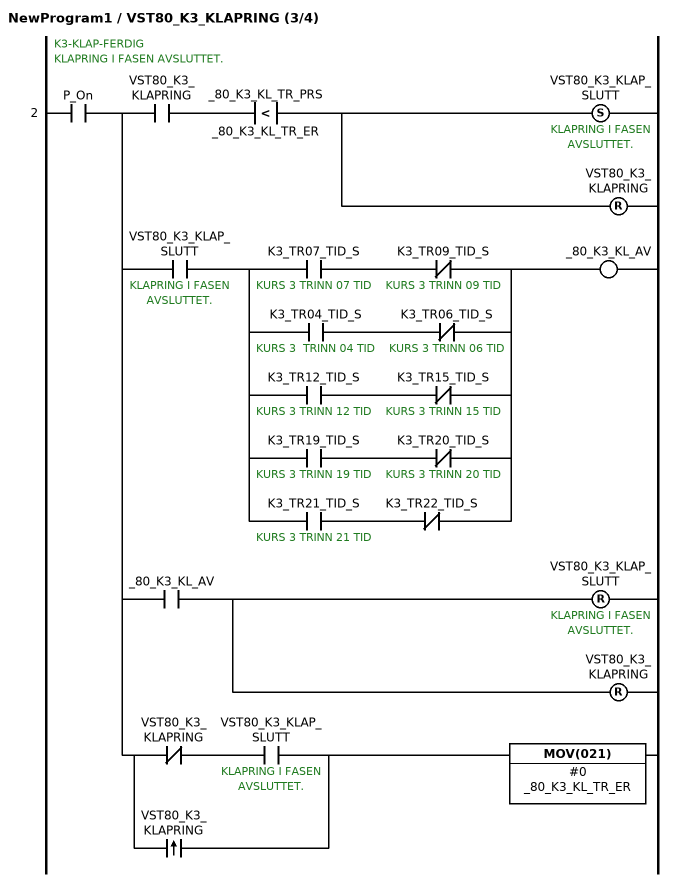
; rung 2: K3-KLAP-FERDIG / KLAPRING I FASEN AVSLUTTET.
LD P_On
OUT TR0
AND VST80_K3_KLAPRING
AND<(310) _80_K3_KL_TR_PRS _80_K3_KL_TR_ER
SET VST80_K3_KLAP_SLUTT  ; KLAPRING I FASEN AVSLUTTET.
RSET VST80_K3_KLAPRING
LD TR0
AND VST80_K3_KLAP_SLUTT  ; KLAPRING I FASEN AVSLUTTET.
LD K3_TR07_TID_S  ; KURS 3 TRINN 07 TID
ANDNOT K3_TR09_TID_S  ; KURS 3 TRINN 09 TID
LD K3_TR04_TID_S  ; KURS 3  TRINN 04 TID
ANDNOT K3_TR06_TID_S  ; KURS 3 TRINN 06 TID
ORLD
LD K3_TR12_TID_S  ; KURS 3 TRINN 12 TID
ANDNOT K3_TR15_TID_S  ; KURS 3 TRINN 15 TID
ORLD
LD K3_TR19_TID_S  ; KURS 3 TRINN 19 TID
ANDNOT K3_TR20_TID_S  ; KURS 3 TRINN 20 TID
ORLD
LD K3_TR21_TID_S  ; KURS 3 TRINN 21 TID
ANDNOT K3_TR22_TID_S
ORLD
ANDLD
OUT _80_K3_KL_AV
LD TR0
AND _80_K3_KL_AV
RSET VST80_K3_KLAP_SLUTT  ; KLAPRING I FASEN AVSLUTTET.
RSET VST80_K3_KLAPRING
LD TR0
LDNOT VST80_K3_KLAPRING
AND VST80_K3_KLAP_SLUTT  ; KLAPRING I FASEN AVSLUTTET.
@OR VST80_K3_KLAPRING
ANDLD
MOV(021) #0 _80_K3_KL_TR_ER

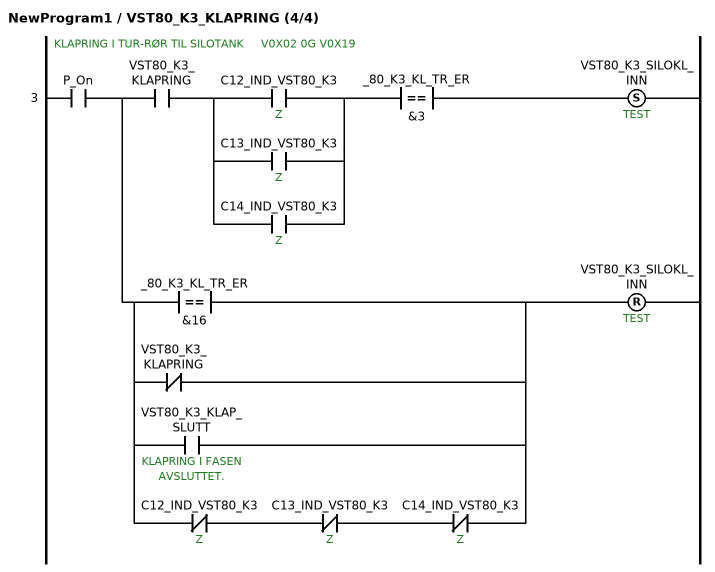
; rung 3: KLAPRING I TUR-RØR TIL SILOTANK     V0X02 0G V0X19
LD P_On
OUT TR0
AND VST80_K3_KLAPRING
LD C12_IND_VST80_K3  ; Z
OR C13_IND_VST80_K3  ; Z
OR C14_IND_VST80_K3  ; Z
ANDLD
AND=(300) _80_K3_KL_TR_ER &3
SET VST80_K3_SILOKL_INN  ; TEST
LD TR0
LD=(300) _80_K3_KL_TR_ER &16
ORNOT VST80_K3_KLAPRING
OR VST80_K3_KLAP_SLUTT  ; KLAPRING I FASEN AVSLUTTET.
LDNOT C12_IND_VST80_K3  ; Z
ANDNOT C13_IND_VST80_K3  ; Z
ANDNOT C14_IND_VST80_K3  ; Z
ORLD
ANDLD
RSET VST80_K3_SILOKL_INN  ; TEST
; rung 4: Ingen_kommentar_funnet

### Section VST80_K3_GRAF_TR_
; OVERFØRING AV TRINN I VASK TIL GRAFIKK

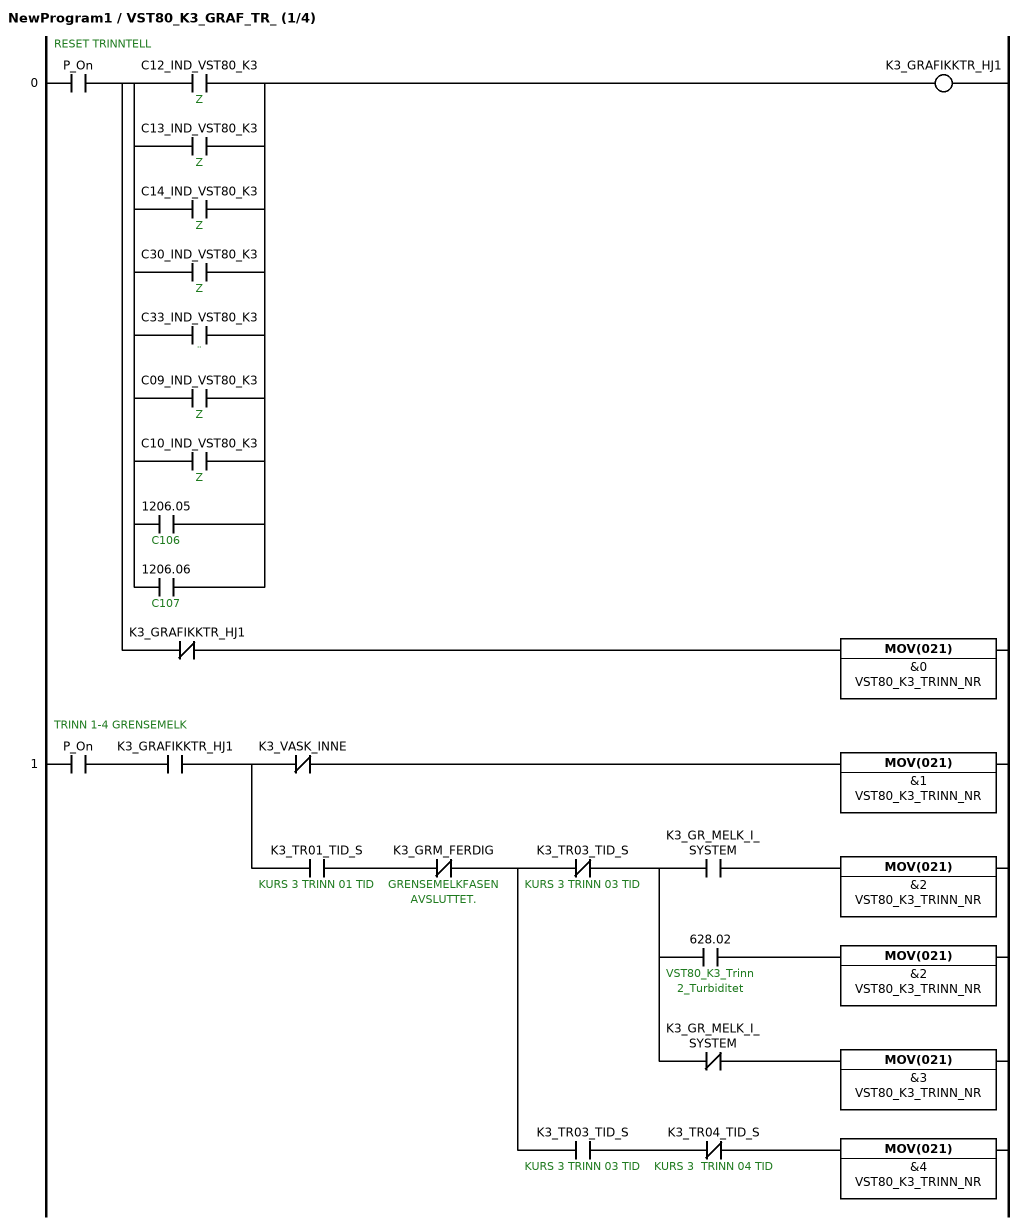
; rung 0: RESET TRINNTELL
LD P_On
OUT TR0
LD C12_IND_VST80_K3  ; Z
OR C13_IND_VST80_K3  ; Z
OR C14_IND_VST80_K3  ; Z
OR C30_IND_VST80_K3  ; Z
OR C33_IND_VST80_K3  ; ¨
OR C09_IND_VST80_K3  ; Z
OR C10_IND_VST80_K3  ; Z
OR 1206.05  ; C106
OR 1206.06  ; C107
ANDLD
OUT K3_GRAFIKKTR_HJ1
LD TR0
ANDNOT K3_GRAFIKKTR_HJ1
MOV(021) &0 VST80_K3_TRINN_NR
; rung 1: TRINN 1-4 GRENSEMELK
LD P_On
AND K3_GRAFIKKTR_HJ1
OUT TR0
ANDNOT K3_VASK_INNE
MOV(021) &1 VST80_K3_TRINN_NR
LD TR0
AND K3_TR01_TID_S  ; KURS 3 TRINN 01 TID
ANDNOT K3_GRM_FERDIG  ; GRENSEMELKFASEN AVSLUTTET.
OUT TR0
ANDNOT K3_TR03_TID_S  ; KURS 3 TRINN 03 TID
OUT TR1
AND K3_GR_MELK_I_SYSTEM
MOV(021) &2 VST80_K3_TRINN_NR
LD TR1
AND 628.02  ; VST80_K3_Trinn 2_Turbiditet
MOV(021) &2 VST80_K3_TRINN_NR
LD TR1
ANDNOT K3_GR_MELK_I_SYSTEM
MOV(021) &3 VST80_K3_TRINN_NR
LD TR0
AND K3_TR03_TID_S  ; KURS 3 TRINN 03 TID
ANDNOT K3_TR04_TID_S  ; KURS 3  TRINN 04 TID
MOV(021) &4 VST80_K3_TRINN_NR

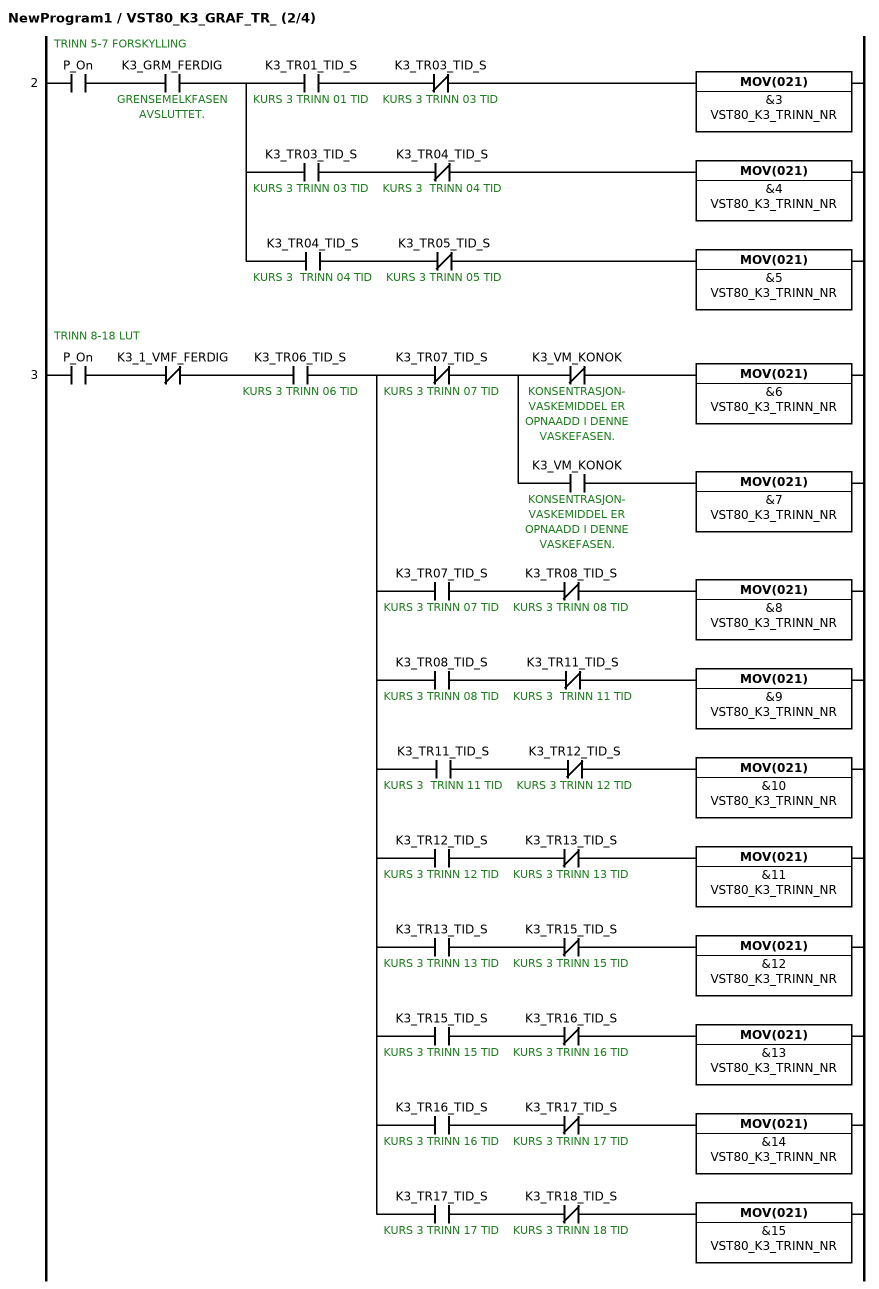
; rung 2: TRINN 5-7 FORSKYLLING
LD P_On
AND K3_GRM_FERDIG  ; GRENSEMELKFASEN AVSLUTTET.
OUT TR0
AND K3_TR01_TID_S  ; KURS 3 TRINN 01 TID
ANDNOT K3_TR03_TID_S  ; KURS 3 TRINN 03 TID
MOV(021) &3 VST80_K3_TRINN_NR
LD TR0
AND K3_TR03_TID_S  ; KURS 3 TRINN 03 TID
ANDNOT K3_TR04_TID_S  ; KURS 3  TRINN 04 TID
MOV(021) &4 VST80_K3_TRINN_NR
LD TR0
AND K3_TR04_TID_S  ; KURS 3  TRINN 04 TID
ANDNOT K3_TR05_TID_S  ; KURS 3 TRINN 05 TID
MOV(021) &5 VST80_K3_TRINN_NR
; rung 3: TRINN 8-18 LUT
LD P_On
ANDNOT K3_1_VMF_FERDIG
AND K3_TR06_TID_S  ; KURS 3 TRINN 06 TID
OUT TR0
ANDNOT K3_TR07_TID_S  ; KURS 3 TRINN 07 TID
OUT TR1
ANDNOT K3_VM_KONOK  ; KONSENTRASJON-VASKEMIDDEL ER OPNAADD I DENNE VASKEFASEN.
MOV(021) &6 VST80_K3_TRINN_NR
LD TR1
AND K3_VM_KONOK  ; KONSENTRASJON-VASKEMIDDEL ER OPNAADD I DENNE VASKEFASEN.
MOV(021) &7 VST80_K3_TRINN_NR
LD TR0
AND K3_TR07_TID_S  ; KURS 3 TRINN 07 TID
ANDNOT K3_TR08_TID_S  ; KURS 3 TRINN 08 TID
MOV(021) &8 VST80_K3_TRINN_NR
LD TR0
AND K3_TR08_TID_S  ; KURS 3 TRINN 08 TID
ANDNOT K3_TR11_TID_S  ; KURS 3  TRINN 11 TID
MOV(021) &9 VST80_K3_TRINN_NR
LD TR0
AND K3_TR11_TID_S  ; KURS 3  TRINN 11 TID
ANDNOT K3_TR12_TID_S  ; KURS 3 TRINN 12 TID
MOV(021) &10 VST80_K3_TRINN_NR
LD TR0
AND K3_TR12_TID_S  ; KURS 3 TRINN 12 TID
ANDNOT K3_TR13_TID_S  ; KURS 3 TRINN 13 TID
MOV(021) &11 VST80_K3_TRINN_NR
LD TR0
AND K3_TR13_TID_S  ; KURS 3 TRINN 13 TID
ANDNOT K3_TR15_TID_S  ; KURS 3 TRINN 15 TID
MOV(021) &12 VST80_K3_TRINN_NR
LD TR0
AND K3_TR15_TID_S  ; KURS 3 TRINN 15 TID
ANDNOT K3_TR16_TID_S  ; KURS 3 TRINN 16 TID
MOV(021) &13 VST80_K3_TRINN_NR
LD TR0
AND K3_TR16_TID_S  ; KURS 3 TRINN 16 TID
ANDNOT K3_TR17_TID_S  ; KURS 3 TRINN 17 TID
MOV(021) &14 VST80_K3_TRINN_NR
LD TR0
AND K3_TR17_TID_S  ; KURS 3 TRINN 17 TID
ANDNOT K3_TR18_TID_S  ; KURS 3 TRINN 18 TID
MOV(021) &15 VST80_K3_TRINN_NR

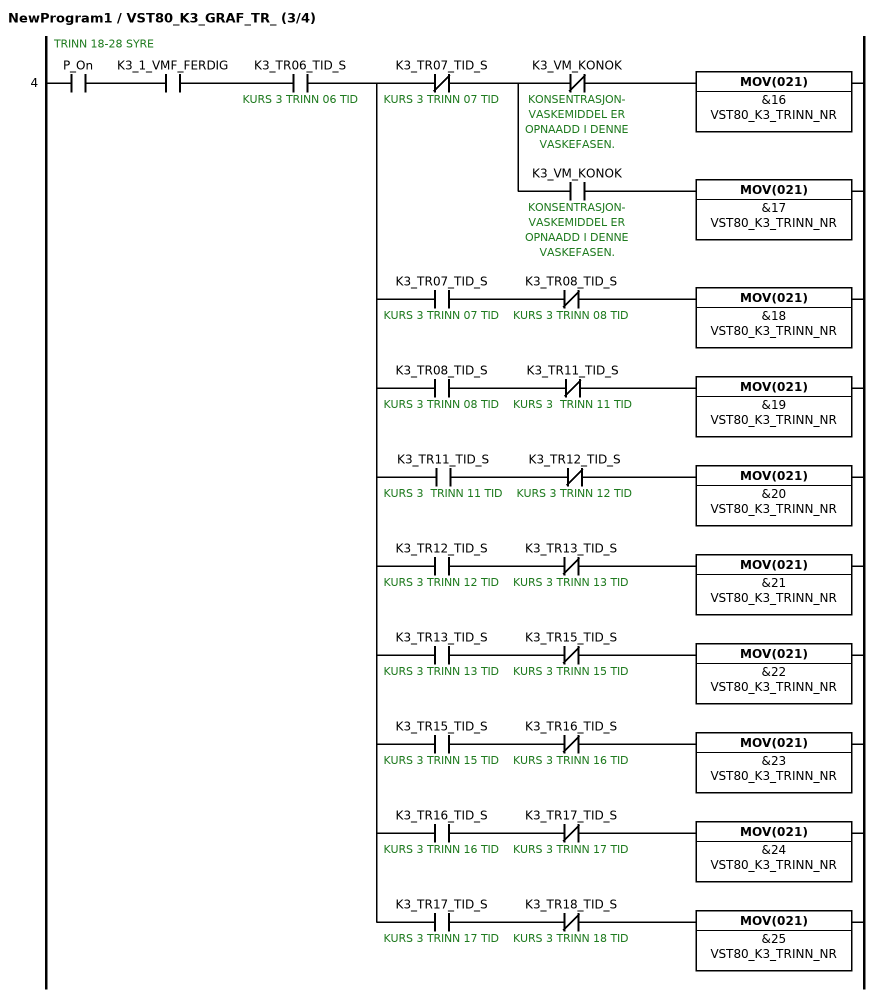
; rung 4: TRINN 18-28 SYRE
LD P_On
AND K3_1_VMF_FERDIG
AND K3_TR06_TID_S  ; KURS 3 TRINN 06 TID
OUT TR0
ANDNOT K3_TR07_TID_S  ; KURS 3 TRINN 07 TID
OUT TR1
ANDNOT K3_VM_KONOK  ; KONSENTRASJON-VASKEMIDDEL ER OPNAADD I DENNE VASKEFASEN.
MOV(021) &16 VST80_K3_TRINN_NR
LD TR1
AND K3_VM_KONOK  ; KONSENTRASJON-VASKEMIDDEL ER OPNAADD I DENNE VASKEFASEN.
MOV(021) &17 VST80_K3_TRINN_NR
LD TR0
AND K3_TR07_TID_S  ; KURS 3 TRINN 07 TID
ANDNOT K3_TR08_TID_S  ; KURS 3 TRINN 08 TID
MOV(021) &18 VST80_K3_TRINN_NR
LD TR0
AND K3_TR08_TID_S  ; KURS 3 TRINN 08 TID
ANDNOT K3_TR11_TID_S  ; KURS 3  TRINN 11 TID
MOV(021) &19 VST80_K3_TRINN_NR
LD TR0
AND K3_TR11_TID_S  ; KURS 3  TRINN 11 TID
ANDNOT K3_TR12_TID_S  ; KURS 3 TRINN 12 TID
MOV(021) &20 VST80_K3_TRINN_NR
LD TR0
AND K3_TR12_TID_S  ; KURS 3 TRINN 12 TID
ANDNOT K3_TR13_TID_S  ; KURS 3 TRINN 13 TID
MOV(021) &21 VST80_K3_TRINN_NR
LD TR0
AND K3_TR13_TID_S  ; KURS 3 TRINN 13 TID
ANDNOT K3_TR15_TID_S  ; KURS 3 TRINN 15 TID
MOV(021) &22 VST80_K3_TRINN_NR
LD TR0
AND K3_TR15_TID_S  ; KURS 3 TRINN 15 TID
ANDNOT K3_TR16_TID_S  ; KURS 3 TRINN 16 TID
MOV(021) &23 VST80_K3_TRINN_NR
LD TR0
AND K3_TR16_TID_S  ; KURS 3 TRINN 16 TID
ANDNOT K3_TR17_TID_S  ; KURS 3 TRINN 17 TID
MOV(021) &24 VST80_K3_TRINN_NR
LD TR0
AND K3_TR17_TID_S  ; KURS 3 TRINN 17 TID
ANDNOT K3_TR18_TID_S  ; KURS 3 TRINN 18 TID
MOV(021) &25 VST80_K3_TRINN_NR

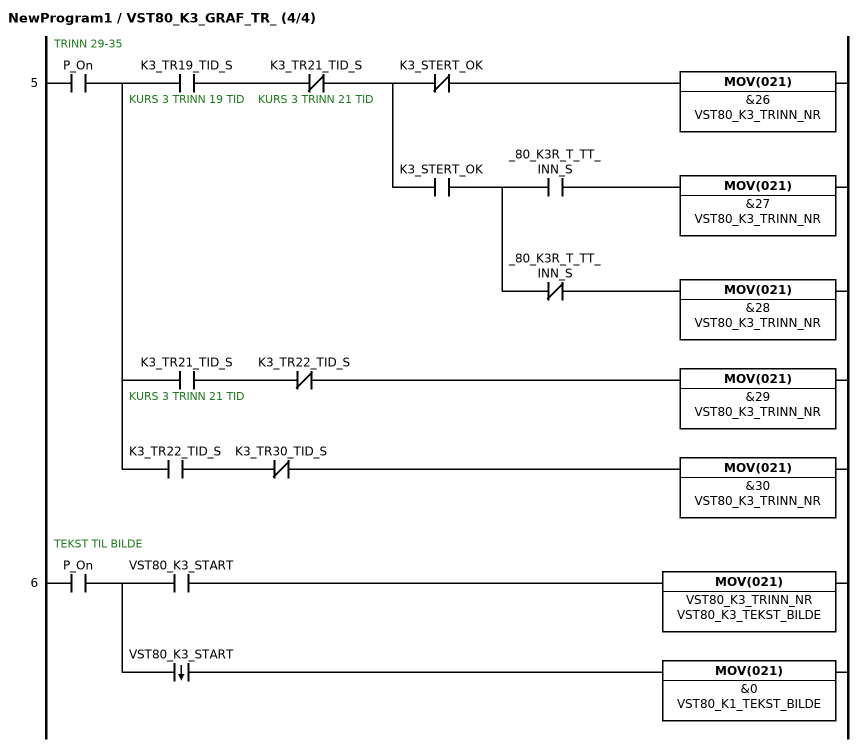
; rung 5: TRINN 29-35
LD P_On
OUT TR0
AND K3_TR19_TID_S  ; KURS 3 TRINN 19 TID
ANDNOT K3_TR21_TID_S  ; KURS 3 TRINN 21 TID
OUT TR1
ANDNOT K3_STERT_OK
MOV(021) &26 VST80_K3_TRINN_NR
LD TR1
AND K3_STERT_OK
OUT TR1
AND _80_K3R_T_TT_INN_S
MOV(021) &27 VST80_K3_TRINN_NR
LD TR1
ANDNOT _80_K3R_T_TT_INN_S
MOV(021) &28 VST80_K3_TRINN_NR
LD TR0
AND K3_TR21_TID_S  ; KURS 3 TRINN 21 TID
ANDNOT K3_TR22_TID_S
MOV(021) &29 VST80_K3_TRINN_NR
LD TR0
AND K3_TR22_TID_S
ANDNOT K3_TR30_TID_S
MOV(021) &30 VST80_K3_TRINN_NR
; rung 6: TEKST TIL BILDE
LD P_On
OUT TR0
AND VST80_K3_START
MOV(021) VST80_K3_TRINN_NR VST80_K3_TEKST_BILDE
LD TR0
%AND VST80_K3_START
MOV(021) &0 VST80_K1_TEKST_BILDE
; rung 7: Ingen_kommentar_funnet

### Section VST80_K3_GRAF_FEIL_TXT

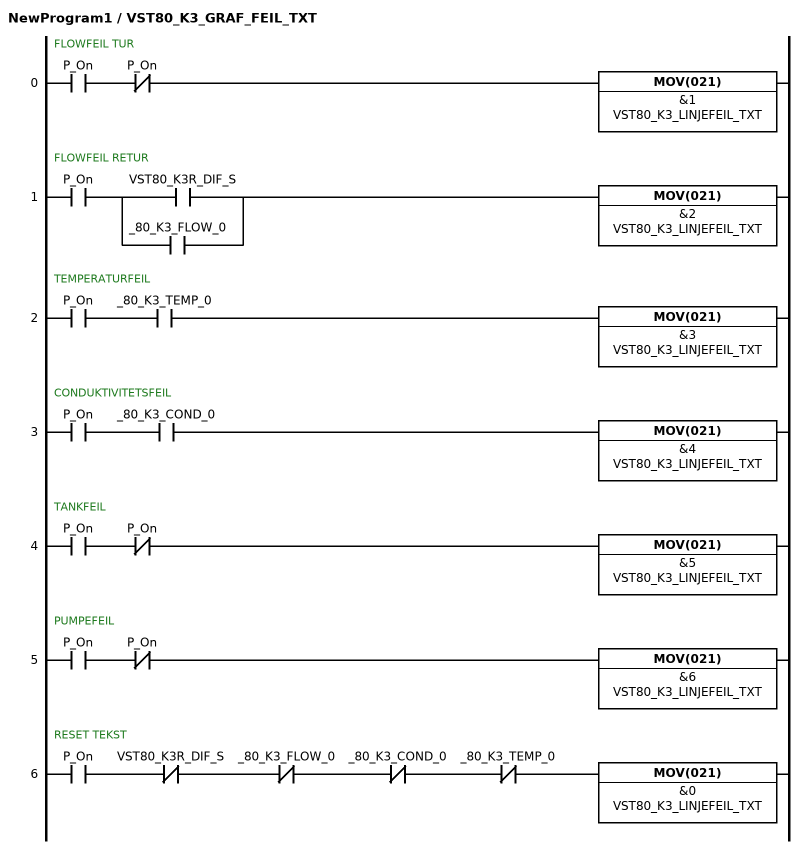
; rung 0: FLOWFEIL TUR
LD P_On
ANDNOT P_On
MOV(021) &1 VST80_K3_LINJEFEIL_TXT
; rung 1: FLOWFEIL RETUR
LD P_On
LD VST80_K3R_DIF_S
OR _80_K3_FLOW_0
ANDLD
MOV(021) &2 VST80_K3_LINJEFEIL_TXT
; rung 2: TEMPERATURFEIL
LD P_On
AND _80_K3_TEMP_0
MOV(021) &3 VST80_K3_LINJEFEIL_TXT
; rung 3: CONDUKTIVITETSFEIL
LD P_On
AND _80_K3_COND_0
MOV(021) &4 VST80_K3_LINJEFEIL_TXT
; rung 4: TANKFEIL
LD P_On
ANDNOT P_On
MOV(021) &5 VST80_K3_LINJEFEIL_TXT
; rung 5: PUMPEFEIL
LD P_On
ANDNOT P_On
MOV(021) &6 VST80_K3_LINJEFEIL_TXT
; rung 6: RESET TEKST
LD P_On
ANDNOT VST80_K3R_DIF_S
ANDNOT _80_K3_FLOW_0
ANDNOT _80_K3_COND_0
ANDNOT _80_K3_TEMP_0
MOV(021) &0 VST80_K3_LINJEFEIL_TXT
; rung 7: Ingen_kommentar_funnet

### Section VST80_K3_TR_VEKS
; VST80 KURS3 VEKSLING AV TRINN.

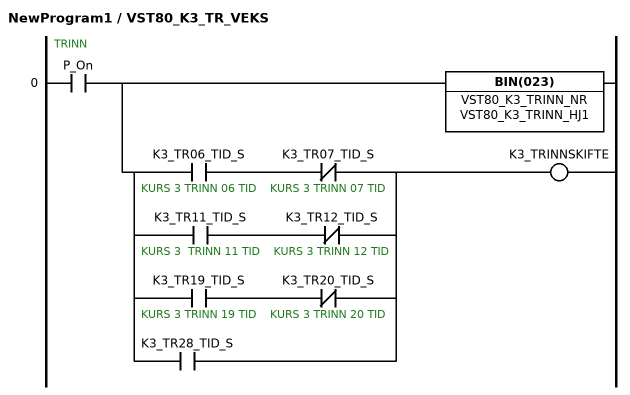
; rung 0: TRINN
LD P_On
BIN(023) VST80_K3_TRINN_NR VST80_K3_TRINN_HJ1
LD K3_TR06_TID_S  ; KURS 3 TRINN 06 TID
ANDNOT K3_TR07_TID_S  ; KURS 3 TRINN 07 TID
LD K3_TR11_TID_S  ; KURS 3  TRINN 11 TID
ANDNOT K3_TR12_TID_S  ; KURS 3 TRINN 12 TID
ORLD
LD K3_TR19_TID_S  ; KURS 3 TRINN 19 TID
ANDNOT K3_TR20_TID_S  ; KURS 3 TRINN 20 TID
ORLD
OR K3_TR28_TID_S
ANDLD
OUT K3_TRINNSKIFTE
; rung 1: Ingen_kommentar_funnet

### Section V80_K3_FEIL_RET
; FEIL I RETUR / FLOW / TEMP / COND

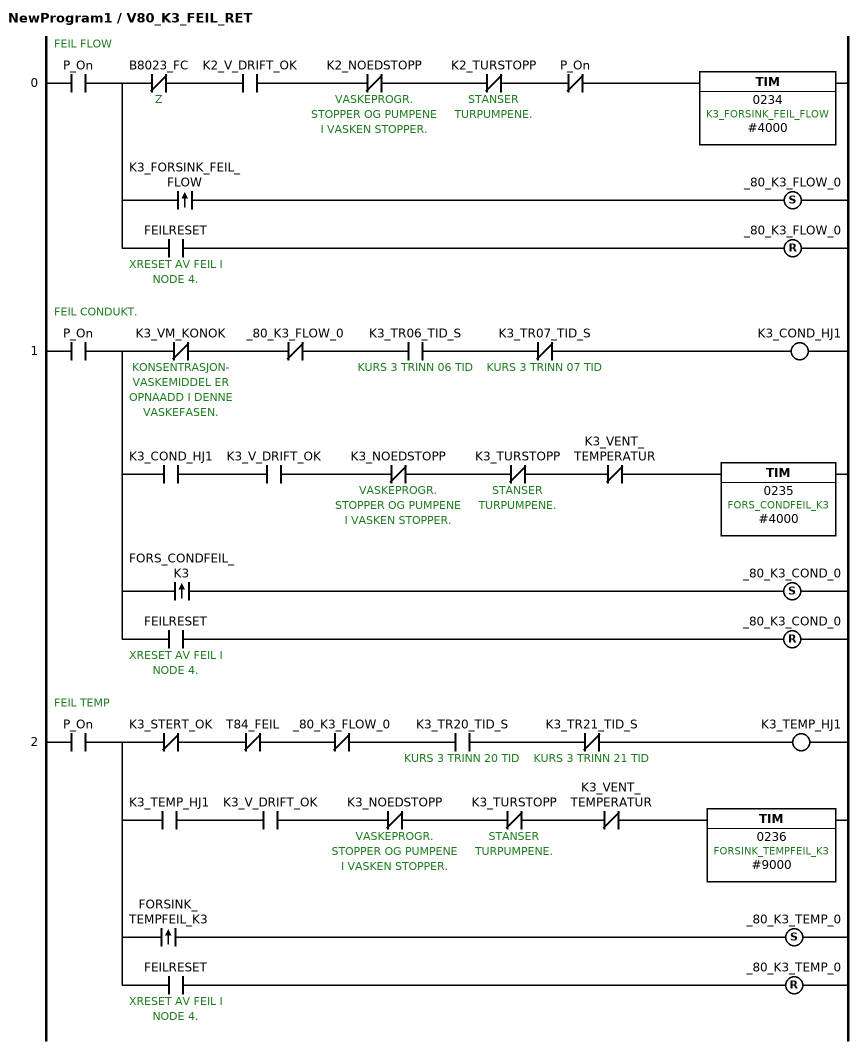
; rung 0: FEIL FLOW
LD P_On
OUT TR0
ANDNOT B8023_FC  ; Z
AND K2_V_DRIFT_OK
ANDNOT K2_NOEDSTOPP  ; VASKEPROGR. STOPPER OG PUMPENE I VASKEN STOPPER.
ANDNOT K2_TURSTOPP  ; STANSER TURPUMPENE.
ANDNOT P_On
TIM 0234 #4000  ; K3_FORSINK_FEIL_FLOW
LD TR0
@AND K3_FORSINK_FEIL_FLOW
SET _80_K3_FLOW_0
LD TR0
AND FEILRESET  ; XRESET AV FEIL I NODE 4.
RSET _80_K3_FLOW_0
; rung 1: FEIL CONDUKT.
LD P_On
OUT TR0
ANDNOT K3_VM_KONOK  ; KONSENTRASJON-VASKEMIDDEL ER OPNAADD I DENNE VASKEFASEN.
ANDNOT _80_K3_FLOW_0
AND K3_TR06_TID_S  ; KURS 3 TRINN 06 TID
ANDNOT K3_TR07_TID_S  ; KURS 3 TRINN 07 TID
OUT K3_COND_HJ1
LD TR0
AND K3_COND_HJ1
AND K3_V_DRIFT_OK
ANDNOT K3_NOEDSTOPP  ; VASKEPROGR. STOPPER OG PUMPENE I VASKEN STOPPER.
ANDNOT K3_TURSTOPP  ; STANSER TURPUMPENE.
ANDNOT K3_VENT_TEMPERATUR
TIM 0235 #4000  ; FORS_CONDFEIL_K3
LD TR0
@AND FORS_CONDFEIL_K3
SET _80_K3_COND_0
LD TR0
AND FEILRESET  ; XRESET AV FEIL I NODE 4.
RSET _80_K3_COND_0
; rung 2: FEIL TEMP
LD P_On
OUT TR0
ANDNOT K3_STERT_OK
ANDNOT T84_FEIL
ANDNOT _80_K3_FLOW_0
AND K3_TR20_TID_S  ; KURS 3 TRINN 20 TID
ANDNOT K3_TR21_TID_S  ; KURS 3 TRINN 21 TID
OUT K3_TEMP_HJ1
LD TR0
AND K3_TEMP_HJ1
AND K3_V_DRIFT_OK
ANDNOT K3_NOEDSTOPP  ; VASKEPROGR. STOPPER OG PUMPENE I VASKEN STOPPER.
ANDNOT K3_TURSTOPP  ; STANSER TURPUMPENE.
ANDNOT K3_VENT_TEMPERATUR
TIM 0236 #9000  ; FORSINK_TEMPFEIL_K3
LD TR0
@AND FORSINK_TEMPFEIL_K3
SET _80_K3_TEMP_0
LD TR0
AND FEILRESET  ; XRESET AV FEIL I NODE 4.
RSET _80_K3_TEMP_0
; rung 3: Ingen_kommentar_funnet

### Section VST80_K3_VASKERAPPORT
; VST80 / KURS3 VASKERAPPORT

